--- Backups/Rob1/HOME/Module1.mod ---
MODULE Module1
!PERS tooldata DrillTool:=[TRUE,[[31.792631019,0,229.638935148],[0.945518576,0,0.325568154,0]],[1,[0,0,1],[1,0,0,0],0,0,0]];
PERS tooldata DrillTool:=[TRUE,[[67.056,0,55.372],[0.7071,0,0.7071,0]],[1,[0,0,1],[1,0,0,0],0,0,0]];
PERS wobjdata FakeWing:=[FALSE, TRUE, "",[[154, -596.9, 290],[0, 0.1326, 0, 0.9912]],[[0, 0, 0],[1, 0, 0, 0]]];
!PERS wobjdata FakeWing:=[FALSE, TRUE, "",[[154, -322.58, 290],[0,0,0,1]],[[0, 0, 0],[1, 0, 0, 0]]];
CONST jointtarget jHome:=[[-90,0,28.434410486,3.185484116,-20,-3.571881577],[9E+09,9E+09,9E+09,9E+09,9E+09,9E+09]];
	CONST robtarget Target_10:=[[25.4,-256.2,-27.8],[0.0113580960105811,-0.801870156996903,0.57220314404859,0.171635680770881],[0,0,0,1],[9E+09,9E+09,9E+09,9E+09,9E+09,9E+09]];
	CONST robtarget Target_20:=[[25.4,-251.5,-26.8],[0.00934854871281768,-0.800936484340026,0.573902636486851,0.170438013727704],[0,0,0,1],[9E+09,9E+09,9E+09,9E+09,9E+09,9E+09]];
	CONST robtarget Target_30:=[[25.4,-246.7,-25.8],[0.00738585622544953,-0.799995428854368,0.575595110655205,0.169242522817864],[0,0,0,1],[9E+09,9E+09,9E+09,9E+09,9E+09,9E+09]];
	CONST robtarget Target_40:=[[25.4,-242,-24.8],[0.00544599211880825,-0.799100144747581,0.577206071085835,0.168054905718017],[0,0,0,1],[9E+09,9E+09,9E+09,9E+09,9E+09,9E+09]];
	CONST robtarget Target_50:=[[25.4,-237.3,-23.8],[0.00347861493687028,-0.798230983744147,0.578772117197483,0.166847331964629],[0,0,0,1],[9E+09,9E+09,9E+09,9E+09,9E+09,9E+09]];
	CONST robtarget Target_60:=[[25.4,-232.5,-22.9],[0.00155774511334554,-0.797353967904281,0.580333117220716,0.165643280438256],[0,0,0,1],[9E+09,9E+09,9E+09,9E+09,9E+09,9E+09]];
	CONST robtarget Target_70:=[[25.4,-227.8,-21.9],[-0.000343161028673128,-0.796523037582201,0.581818895966585,0.164431460303543],[0,0,0,1],[9E+09,9E+09,9E+09,9E+09,9E+09,9E+09]];
	CONST robtarget Target_80:=[[25.4,-223,-21],[-0.00227982923064156,-0.795692138630642,0.58329634877276,0.163199854192462],[0,0,0,1],[9E+09,9E+09,9E+09,9E+09,9E+09,9E+09]];
	CONST robtarget Target_90:=[[25.4,-218.3,-20.1],[-0.00415671334714131,-0.794897215588351,0.584705500460769,0.161989555573681],[0,0,0,1],[9E+09,9E+09,9E+09,9E+09,9E+09,9E+09]];
	CONST robtarget Target_100:=[[25.4,-213.5,-19.2],[-0.00606983909444402,-0.794105676665045,0.586106608579309,0.160743194945786],[0,0,0,1],[9E+09,9E+09,9E+09,9E+09,9E+09,9E+09]];
	CONST robtarget Target_110:=[[25.4,-208.8,-18.4],[-0.00792422315599783,-0.793348049062693,0.587443386601589,0.159519112566011],[0,0,0,1],[9E+09,9E+09,9E+09,9E+09,9E+09,9E+09]];
	CONST robtarget Target_120:=[[25.4,-204,-17.6],[-0.00977383985694139,-0.792585828477493,0.588775847716777,0.158288274033445],[0,0,0,1],[9E+09,9E+09,9E+09,9E+09,9E+09,9E+09]];
	CONST robtarget Target_130:=[[25.4,-199.3,-16.8],[-0.0116479972262109,-0.79187063814985,0.590041679393542,0.157022397049646],[0,0,0,1],[9E+09,9E+09,9E+09,9E+09,9E+09,9E+09]];
	CONST robtarget Target_140:=[[25.4,-194.5,-16],[-0.0134775760488848,-0.791139740266602,0.591307245188397,0.155794762756806],[0,0,0,1],[9E+09,9E+09,9E+09,9E+09,9E+09,9E+09]];
	CONST robtarget Target_150:=[[25.4,-189.8,-15.2],[-0.0152917657314588,-0.790446591060719,0.592512479634857,0.154561670728084],[0,0,0,1],[9E+09,9E+09,9E+09,9E+09,9E+09,9E+09]];
	CONST robtarget Target_160:=[[25.4,-185.1,-14.4],[-0.0170965714657476,-0.789768956804693,0.593687446554438,0.153322920385096],[0,0,0,1],[9E+09,9E+09,9E+09,9E+09,9E+09,9E+09]];
	CONST robtarget Target_170:=[[25.4,-180.3,-13.7],[-0.0189383920181083,-0.7890933742209,0.594856495857871,0.152048457421108],[0,0,0,1],[9E+09,9E+09,9E+09,9E+09,9E+09,9E+09]];
	CONST robtarget Target_180:=[[25.4,-175.6,-13],[-0.0207248929133501,-0.788445598386254,0.595972909516474,0.150798900266347],[0,0,0,1],[9E+09,9E+09,9E+09,9E+09,9E+09,9E+09]];
	CONST robtarget Target_190:=[[25.4,-170.8,-12.3],[-0.0225484722456159,-0.787799513101417,0.597083852612889,0.149513766943077],[0,0,0,1],[9E+09,9E+09,9E+09,9E+09,9E+09,9E+09]];
	CONST robtarget Target_200:=[[25.4,-166.1,-11.6],[-0.0243197129064465,-0.787176744880257,0.598145161875128,0.148268975882507],[0,0,0,1],[9E+09,9E+09,9E+09,9E+09,9E+09,9E+09]];
	CONST robtarget Target_210:=[[25.4,-161.3,-11],[-0.0260874898804154,-0.78654858525833,0.5992047460239,0.147018496259117],[0,0,0,1],[9E+09,9E+09,9E+09,9E+09,9E+09,9E+09]];
	CONST robtarget Target_220:=[[25.4,-156.6,-10.3],[-0.0278809945750648,-0.78596193798026,0.600210217810398,0.145719513531353],[0,0,0,1],[9E+09,9E+09,9E+09,9E+09,9E+09,9E+09]];
	CONST robtarget Target_230:=[[25.4,-151.8,-9.7],[-0.0296325952340913,-0.785359970763115,0.601217933569803,0.144459759022046],[0,0,0,1],[9E+09,9E+09,9E+09,9E+09,9E+09,9E+09]];
	CONST robtarget Target_240:=[[25.4,-147.1,-9.1],[-0.0313751328555289,-0.784785659070614,0.602177510654819,0.143210739879962],[0,0,0,1],[9E+09,9E+09,9E+09,9E+09,9E+09,9E+09]];
	CONST robtarget Target_250:=[[25.4,-142.3,-8.5],[-0.0331524140005,-0.784214983247709,0.603132486603527,0.1419118779355],[0,0,0,1],[9E+09,9E+09,9E+09,9E+09,9E+09,9E+09]];
	CONST robtarget Target_260:=[[25.4,-137.6,-8],[-0.034877347640361,-0.783666646083767,0.604045100801052,0.140640231212982],[0,0,0,1],[9E+09,9E+09,9E+09,9E+09,9E+09,9E+09]];
	CONST robtarget Target_270:=[[25.4,-132.9,-7.4],[-0.0365986103919072,-0.783126667075213,0.604935351521993,0.139378569055698],[0,0,0,1],[9E+09,9E+09,9E+09,9E+09,9E+09,9E+09]];
	CONST robtarget Target_280:=[[25.4,-128.1,-6.9],[-0.0383577272294432,-0.782587224758595,0.605821324762428,0.138081290801936],[0,0,0,1],[9E+09,9E+09,9E+09,9E+09,9E+09,9E+09]];
	CONST robtarget Target_290:=[[25.4,-123.4,-6.4],[-0.0400656367387652,-0.782068484600279,0.606668087171559,0.136811776376679],[0,0,0,1],[9E+09,9E+09,9E+09,9E+09,9E+09,9E+09]];
	CONST robtarget Target_300:=[[25.4,-118.6,-5.9],[-0.0417706616179563,-0.781543829458959,0.607514638958406,0.135537514784141],[0,0,0,1],[9E+09,9E+09,9E+09,9E+09,9E+09,9E+09]];
	CONST robtarget Target_310:=[[25.4,-113.9,-5.4],[-0.0435063932859472,-0.781051177343454,0.608316177335671,0.134229953830614],[0,0,0,1],[9E+09,9E+09,9E+09,9E+09,9E+09,9E+09]];
	CONST robtarget Target_320:=[[25.4,-109.1,-5],[-0.0452028740439187,-0.780544008668363,0.609121417468522,0.132961834716695],[0,0,0,1],[9E+09,9E+09,9E+09,9E+09,9E+09,9E+09]];
	CONST robtarget Target_330:=[[25.4,-104.4,-4.6],[-0.046885611949136,-0.780063932790252,0.609887552842283,0.131678293731398],[0,0,0,1],[9E+09,9E+09,9E+09,9E+09,9E+09,9E+09]];
	CONST robtarget Target_340:=[[25.4,-99.6,-4.2],[-0.04861077072326,-0.779581431143657,0.610649531901286,0.130372291436634],[0,0,0,1],[9E+09,9E+09,9E+09,9E+09,9E+09,9E+09]];
	CONST robtarget Target_350:=[[25.4,-94.9,-3.8],[-0.0502864189787529,-0.779116692721743,0.611377853226394,0.129095219791102],[0,0,0,1],[9E+09,9E+09,9E+09,9E+09,9E+09,9E+09]];
	CONST robtarget Target_360:=[[25.4,-90.1,-3.4],[-0.0520001006783575,-0.778651616514941,0.612102328073387,0.127782587214575],[0,0,0,1],[9E+09,9E+09,9E+09,9E+09,9E+09,9E+09]];
	CONST robtarget Target_370:=[[25.4,-85.4,-3.1],[-0.0536646621305004,-0.778203412489929,0.612794807637811,0.126499314462914],[0,0,0,1],[9E+09,9E+09,9E+09,9E+09,9E+09,9E+09]];
	CONST robtarget Target_380:=[[25.4,-80.7,-2.7],[-0.0553238489574246,-0.77776300170738,0.613470169447094,0.125213162687542],[0,0,0,1],[9E+09,9E+09,9E+09,9E+09,9E+09,9E+09]];
	CONST robtarget Target_390:=[[25.4,-75.9,-2.4],[-0.0569860150022066,-0.77731443415222,0.614145686708351,0.123935225219912],[0,0,0,1],[9E+09,9E+09,9E+09,9E+09,9E+09,9E+09]];
	CONST robtarget Target_400:=[[25.4,-71.2,-2.1],[-0.0586751876109112,-0.776894569887548,0.614783164526675,0.122612031435063],[0,0,0,1],[9E+09,9E+09,9E+09,9E+09,9E+09,9E+09]];
	CONST robtarget Target_410:=[[25.4,-66.4,-1.9],[-0.0603271872625083,-0.776461071687208,0.615425263134368,0.121328397860276],[0,0,0,1],[9E+09,9E+09,9E+09,9E+09,9E+09,9E+09]];
	CONST robtarget Target_420:=[[25.4,-61.7,-1.6],[-0.0619717124676495,-0.776047982126195,0.616034600462907,0.120043356018546],[0,0,0,1],[9E+09,9E+09,9E+09,9E+09,9E+09,9E+09]];
	CONST robtarget Target_430:=[[25.4,-56.9,-1.4],[-0.063654337047,-0.775633930210214,0.616640125167891,0.118722734615959],[0,0,0,1],[9E+09,9E+09,9E+09,9E+09,9E+09,9E+09]];
	CONST robtarget Target_440:=[[25.4,-52.2,-1.1],[-0.0652893578640036,-0.775234130977816,0.61721871302553,0.117432543223271],[0,0,0,1],[9E+09,9E+09,9E+09,9E+09,9E+09,9E+09]];
	CONST robtarget Target_450:=[[25.4,-47.4,-0.9],[-0.0669689070708674,-0.774831453886875,0.617792784809483,0.116118295675694],[0,0,0,1],[9E+09,9E+09,9E+09,9E+09,9E+09,9E+09]];
	CONST robtarget Target_460:=[[25.4,-42.7,-0.8],[-0.0685947840793333,-0.774444127586446,0.618341874516178,0.114823233989456],[0,0,0,1],[9E+09,9E+09,9E+09,9E+09,9E+09,9E+09]];
	CONST robtarget Target_470:=[[25.4,-37.9,-0.6],[-0.0702251950846496,-0.774048910249563,0.618891208798363,0.113535801353087],[0,0,0,1],[9E+09,9E+09,9E+09,9E+09,9E+09,9E+09]];
	CONST robtarget Target_480:=[[25.4,-33.2,-0.5],[-0.0718893502838438,-0.773676551204279,0.619406337541587,0.112215437644457],[0,0,0,1],[9E+09,9E+09,9E+09,9E+09,9E+09,9E+09]];
	CONST robtarget Target_490:=[[25.4,-28.5,-0.3],[-0.0735091429764661,-0.773304826213177,0.619912706592075,0.110924694545269],[0,0,0,1],[9E+09,9E+09,9E+09,9E+09,9E+09,9E+09]];
	CONST robtarget Target_500:=[[25.4,-23.7,-0.2],[-0.0751268762924455,-0.772926904927033,0.620420125378589,0.109630379565486],[0,0,0,1],[9E+09,9E+09,9E+09,9E+09,9E+09,9E+09]];
	CONST robtarget Target_510:=[[25.4,-19,-0.2],[-0.0767785359193531,-0.772570517222499,0.620894717021794,0.108303290416625],[0,0,0,1],[9E+09,9E+09,9E+09,9E+09,9E+09,9E+09]];
	CONST robtarget Target_520:=[[25.4,-14.2,-0.1],[-0.0783956408178687,-0.772201769929318,0.621374495212959,0.107015357391473],[0,0,0,1],[9E+09,9E+09,9E+09,9E+09,9E+09,9E+09]];
	CONST robtarget Target_530:=[[25.4,-9.5,0],[-0.0799992230274888,-0.771850747246867,0.621828447919395,0.105716269550184],[0,0,0,1],[9E+09,9E+09,9E+09,9E+09,9E+09,9E+09]];
	CONST robtarget Target_540:=[[25.4,-4.7,0],[-0.0816486492100062,-0.771496504751779,0.622277235046125,0.104391972782008],[0,0,0,1],[9E+09,9E+09,9E+09,9E+09,9E+09,9E+09]];
	CONST robtarget Target_550:=[[25.4,0,0],[-0.0832525257048043,-0.77115343963232,0.622705329863117,0.103099280633186],[0,0,0,1],[9E+09,9E+09,9E+09,9E+09,9E+09,9E+09]];
	CONST robtarget Target_560:=[[30.1,0,-1.3],[-0.0836404536862687,-0.768801362660341,0.625606921371793,0.102784819941782],[0,0,0,1],[9E+09,9E+09,9E+09,9E+09,9E+09,9E+09]];
	CONST robtarget Target_570:=[[34.8,0,-2.6],[-0.0840284058612932,-0.766430934306805,0.628508693841452,0.102467905764289],[0,0,0,1],[9E+09,9E+09,9E+09,9E+09,9E+09,9E+09]];
	CONST robtarget Target_580:=[[39.5,0,-3.9],[-0.0844163267896941,-0.764042324397513,0.631410232595209,0.10214856080555],[0,0,0,1],[9E+09,9E+09,9E+09,9E+09,9E+09,9E+09]];
	CONST robtarget Target_590:=[[44.2,0,-5.1],[-0.0848041606261163,-0.761635712421235,0.634311119925615,0.101826809062296],[0,0,0,1],[9E+09,9E+09,9E+09,9E+09,9E+09,9E+09]];
	CONST robtarget Target_600:=[[49,0,-6.4],[-0.085200097924907,-0.759159511925291,0.637272618861068,0.101495753688988],[0,0,0,1],[9E+09,9E+09,9E+09,9E+09,9E+09,9E+09]];
	CONST robtarget Target_610:=[[53.7,0,-7.7],[-0.0855875837551199,-0.756717100367288,0.640170903203522,0.101169215724299],[0,0,0,1],[9E+09,9E+09,9E+09,9E+09,9E+09,9E+09]];
	CONST robtarget Target_620:=[[58.4,0,-9],[-0.0859748117230649,-0.754257287630898,0.643067258809194,0.100840351310837],[0,0,0,1],[9E+09,9E+09,9E+09,9E+09,9E+09,9E+09]];
	CONST robtarget Target_630:=[[63.1,0,-10.3],[-0.0863617247713559,-0.751780291900885,0.645961258904983,0.100509189618791],[0,0,0,1],[9E+09,9E+09,9E+09,9E+09,9E+09,9E+09]];
	CONST robtarget Target_640:=[[67.8,0,-11.6],[-0.0867482656496363,-0.7492863408784,0.648852475274426,0.100175761090643],[0,0,0,1],[9E+09,9E+09,9E+09,9E+09,9E+09,9E+09]];
	CONST robtarget Target_650:=[[72.6,0,-12.8],[-0.087142587005737,-0.746722073369839,0.651801887415907,0.0998329316070456],[0,0,0,1],[9E+09,9E+09,9E+09,9E+09,9E+09,9E+09]];
	CONST robtarget Target_660:=[[77.3,0,-14.1],[-0.0875282002573034,-0.744194584856974,0.654686165400069,0.0994950192875346],[0,0,0,1],[9E+09,9E+09,9E+09,9E+09,9E+09,9E+09]];
	CONST robtarget Target_670:=[[82,0,-15.4],[-0.0879132676563278,-0.741650886033532,0.657566360561706,0.0991549397322007],[0,0,0,1],[9E+09,9E+09,9E+09,9E+09,9E+09,9E+09]];
	CONST robtarget Target_680:=[[86.7,0,-16.7],[-0.0882977316351558,-0.739091242029488,0.660442042311056,0.098812728387569],[0,0,0,1],[9E+09,9E+09,9E+09,9E+09,9E+09,9E+09]];
	CONST robtarget Target_690:=[[91.4,0,-18],[-0.0886815346640349,-0.736515927004876,0.663312780341852,0.0984684219074372],[0,0,0,1],[9E+09,9E+09,9E+09,9E+09,9E+09,9E+09]];
	CONST robtarget Target_700:=[[96.1,0,-19.3],[-0.0890646192984286,-0.73392522401178,0.66617814498522,0.098122058134425],[0,0,0,1],[9E+09,9E+09,9E+09,9E+09,9E+09,9E+09]];
	CONST robtarget Target_710:=[[100.9,0,-20.5],[-0.0894550536127219,-0.73126382047628,0.669098483154106,0.097766242059591],[0,0,0,1],[9E+09,9E+09,9E+09,9E+09,9E+09,9E+09]];
	CONST robtarget Target_720:=[[105.6,0,-21.8],[-0.0898365113642169,-0.728642914020408,0.671951679173837,0.0974158402376966],[0,0,0,1],[9E+09,9E+09,9E+09,9E+09,9E+09,9E+09]];
	CONST robtarget Target_730:=[[110.3,0,-23.1],[-0.0902170781671603,-0.726007527181841,0.674798211150562,0.0970635024625115],[0,0,0,1],[9E+09,9E+09,9E+09,9E+09,9E+09,9E+09]];
	CONST robtarget Target_740:=[[115,0,-24.4],[-0.0905966974007335,-0.72335797710495,0.677637655576582,0.0967092711346199],[0,0,0,1],[9E+09,9E+09,9E+09,9E+09,9E+09,9E+09]];
	CONST robtarget Target_750:=[[119.7,0,-25.7],[-0.0909753127685873,-0.720694588932015,0.680469591371138,0.0963531897238861],[0,0,0,1],[9E+09,9E+09,9E+09,9E+09,9E+09,9E+09]];
	CONST robtarget Target_760:=[[119.7,-4.7,-25.7],[-0.0894964456603955,-0.720663942150709,0.680499152895289,0.097748512043658],[0,0,0,1],[9E+09,9E+09,9E+09,9E+09,9E+09,9E+09]];
	CONST robtarget Target_770:=[[119.7,-9.4,-25.7],[-0.0880162719808697,-0.720632874639458,0.680523367054942,0.0991430418519903],[0,0,0,1],[9E+09,9E+09,9E+09,9E+09,9E+09,9E+09]];
	CONST robtarget Target_780:=[[119.7,-14.2,-25.8],[-0.0865428018846856,-0.720603495890162,0.680537461381074,0.100547047742977],[0,0,0,1],[9E+09,9E+09,9E+09,9E+09,9E+09,9E+09]];
	CONST robtarget Target_790:=[[119.7,-18.9,-25.8],[-0.085059938553443,-0.720571800799192,0.680550756587509,0.101939955142535],[0,0,0,1],[9E+09,9E+09,9E+09,9E+09,9E+09,9E+09]];
	CONST robtarget Target_800:=[[119.7,-23.6,-25.9],[-0.083584041621182,-0.720538427344595,0.680557491801351,0.103342068196353],[0,0,0,1],[9E+09,9E+09,9E+09,9E+09,9E+09,9E+09]];
	CONST robtarget Target_810:=[[119.7,-28.3,-26],[-0.0821066527591594,-0.720504826362092,0.680558671847999,0.104743433847213],[0,0,0,1],[9E+09,9E+09,9E+09,9E+09,9E+09,9E+09]];
	CONST robtarget Target_820:=[[119.7,-33.1,-26.2],[-0.0806272283124645,-0.720474728202172,0.680550348761864,0.106144424614581],[0,0,0,1],[9E+09,9E+09,9E+09,9E+09,9E+09,9E+09]];
	CONST robtarget Target_830:=[[119.7,-37.8,-26.3],[-0.0791469179971094,-0.720440954411049,0.680540124134773,0.107544111979611],[0,0,0,1],[9E+09,9E+09,9E+09,9E+09,9E+09,9E+09]];
	CONST robtarget Target_840:=[[119.7,-42.5,-26.5],[-0.0776727785581285,-0.720405551888667,0.680523246637386,0.108953618871318],[0,0,0,1],[9E+09,9E+09,9E+09,9E+09,9E+09,9E+09]];
	CONST robtarget Target_850:=[[119.7,-47.2,-26.6],[-0.0761895130311405,-0.720371815338409,0.680501393526366,0.110351525493748],[0,0,0,1],[9E+09,9E+09,9E+09,9E+09,9E+09,9E+09]];
	CONST robtarget Target_860:=[[119.7,-52,-26.8],[-0.0747115228913701,-0.720340440006396,0.680468644477677,0.111759843957285],[0,0,0,1],[9E+09,9E+09,9E+09,9E+09,9E+09,9E+09]];
	CONST robtarget Target_870:=[[119.7,-56.7,-27.1],[-0.0732253755943593,-0.720307140577433,0.680434751151304,0.113155720261464],[0,0,0,1],[9E+09,9E+09,9E+09,9E+09,9E+09,9E+09]];
	CONST robtarget Target_880:=[[119.7,-61.4,-27.3],[-0.0717448887914529,-0.720272374985656,0.68039399227409,0.114561738997581],[0,0,0,1],[9E+09,9E+09,9E+09,9E+09,9E+09,9E+09]];
	CONST robtarget Target_890:=[[119.7,-66.1,-27.6],[-0.0702696329912503,-0.720236097011316,0.680346371155896,0.1159782673443],[0,0,0,1],[9E+09,9E+09,9E+09,9E+09,9E+09,9E+09]];
	CONST robtarget Target_900:=[[119.7,-70.9,-27.8],[-0.0687850809253925,-0.720206259937601,0.680288774358502,0.117382874690421],[0,0,0,1],[9E+09,9E+09,9E+09,9E+09,9E+09,9E+09]];
	CONST robtarget Target_910:=[[119.7,-75.6,-28.1],[-0.0672996627808184,-0.720172832813,0.680229181677042,0.118785969974019],[0,0,0,1],[9E+09,9E+09,9E+09,9E+09,9E+09,9E+09]];
	CONST robtarget Target_920:=[[119.7,-80.3,-28.4],[-0.0658190780270005,-0.720138044734531,0.680162517796056,0.120199812308221],[0,0,0,1],[9E+09,9E+09,9E+09,9E+09,9E+09,9E+09]];
	CONST robtarget Target_930:=[[119.7,-85,-28.8],[-0.064336655652234,-0.720103899683729,0.680089342195864,0.121612725614418],[0,0,0,1],[9E+09,9E+09,9E+09,9E+09,9E+09,9E+09]];
	CONST robtarget Target_940:=[[119.7,-89.8,-29.1],[-0.0628515923557622,-0.72007501831515,0.680004764514919,0.123025060755081],[0,0,0,1],[9E+09,9E+09,9E+09,9E+09,9E+09,9E+09]];
	CONST robtarget Target_950:=[[119.7,-94.5,-29.5],[-0.0613655083938046,-0.720042568279418,0.67991814027433,0.124435914313536],[0,0,0,1],[9E+09,9E+09,9E+09,9E+09,9E+09,9E+09]];
	CONST robtarget Target_960:=[[119.7,-99.2,-29.9],[-0.0598776216216156,-0.720011096866214,0.679824658385715,0.125845638260513],[0,0,0,1],[9E+09,9E+09,9E+09,9E+09,9E+09,9E+09]];
	CONST robtarget Target_970:=[[119.7,-103.9,-30.3],[-0.058387940861709,-0.719980723710131,0.679724196561222,0.127254164792231],[0,0,0,1],[9E+09,9E+09,9E+09,9E+09,9E+09,9E+09]];
	CONST robtarget Target_980:=[[119.7,-108.6,-30.7],[-0.0569019629309244,-0.719949270323902,0.679616191781681,0.12867418794325],[0,0,0,1],[9E+09,9E+09,9E+09,9E+09,9E+09,9E+09]];
	CONST robtarget Target_990:=[[119.7,-113.4,-31.2],[-0.0554129551896327,-0.719924020676598,0.679495748554978,0.130093568425584],[0,0,0,1],[9E+09,9E+09,9E+09,9E+09,9E+09,9E+09]];
	CONST robtarget Target_1000:=[[119.7,-118.1,-31.7],[-0.0539227905908445,-0.719895285225862,0.679373134873898,0.131511423747453],[0,0,0,1],[9E+09,9E+09,9E+09,9E+09,9E+09,9E+09]];
	CONST robtarget Target_1010:=[[119.7,-122.8,-32.2],[-0.0524305493384612,-0.7198680665055,0.679243054579513,0.132928090060728],[0,0,0,1],[9E+09,9E+09,9E+09,9E+09,9E+09,9E+09]];
	CONST robtarget Target_1020:=[[119.7,-127.5,-32.7],[-0.0509362308012004,-0.719842507181339,0.6791053603599,0.134343495477456],[0,0,0,1],[9E+09,9E+09,9E+09,9E+09,9E+09,9E+09]];
	CONST robtarget Target_1030:=[[119.7,-132.3,-33.2],[-0.0494387596832467,-0.71982411965525,0.678954212481979,0.135757957985906],[0,0,0,1],[9E+09,9E+09,9E+09,9E+09,9E+09,9E+09]];
	CONST robtarget Target_1040:=[[119.7,-137,-33.7],[-0.0479448372699026,-0.719799803937581,0.67880042479814,0.137184248820506],[0,0,0,1],[9E+09,9E+09,9E+09,9E+09,9E+09,9E+09]];
	CONST robtarget Target_1050:=[[119.7,-141.7,-34.3],[-0.0464440772866591,-0.719780190794116,0.678638852589163,0.138595571292312],[0,0,0,1],[9E+09,9E+09,9E+09,9E+09,9E+09,9E+09]];
	CONST robtarget Target_1060:=[[119.7,-146.4,-34.9],[-0.044945509749326,-0.719760119267005,0.678468776104705,0.140019254808413],[0,0,0,1],[9E+09,9E+09,9E+09,9E+09,9E+09,9E+09]];
	CONST robtarget Target_1070:=[[119.7,-151.2,-35.5],[-0.04344331380953,-0.719748215733065,0.67828412552036,0.141441965135516],[0,0,0,1],[9E+09,9E+09,9E+09,9E+09,9E+09,9E+09]];
	CONST robtarget Target_1080:=[[119.7,-155.9,-36.1],[-0.0419398630139701,-0.719733141246756,0.678096934583651,0.142862873377593],[0,0,0,1],[9E+09,9E+09,9E+09,9E+09,9E+09,9E+09]];
	CONST robtarget Target_1090:=[[119.7,-160.6,-36.8],[-0.0404378111769494,-0.719717853139121,0.677900787346707,0.144296631335408],[0,0,0,1],[9E+09,9E+09,9E+09,9E+09,9E+09,9E+09]];
	CONST robtarget Target_1100:=[[119.7,-165.3,-37.4],[-0.0389292896217268,-0.719708346409807,0.677695848544467,0.145714595642316],[0,0,0,1],[9E+09,9E+09,9E+09,9E+09,9E+09,9E+09]];
	CONST robtarget Target_1110:=[[119.7,-170.1,-38.1],[-0.0374204463715451,-0.719705234895391,0.677474850520684,0.147145886689034],[0,0,0,1],[9E+09,9E+09,9E+09,9E+09,9E+09,9E+09]];
	CONST robtarget Target_1120:=[[119.7,-174.8,-38.8],[-0.0359101121108122,-0.719699125713495,0.677251057216981,0.148575360655468],[0,0,0,1],[9E+09,9E+09,9E+09,9E+09,9E+09,9E+09]];
	CONST robtarget Target_1130:=[[119.7,-179.5,-39.6],[-0.0343969212798386,-0.719696439264827,0.677017651592734,0.150003288456814],[0,0,0,1],[9E+09,9E+09,9E+09,9E+09,9E+09,9E+09]];
	CONST robtarget Target_1140:=[[119.7,-184.2,-40.3],[-0.0328808379407684,-0.719697403969569,0.676774392615492,0.151429583357108],[0,0,0,1],[9E+09,9E+09,9E+09,9E+09,9E+09,9E+09]];
	CONST robtarget Target_1150:=[[119.7,-189,-41.1],[-0.0313227011217989,-0.719701525474739,0.676515916078243,0.152888253036598],[0,0,0,1],[9E+09,9E+09,9E+09,9E+09,9E+09,9E+09]];
	CONST robtarget Target_1160:=[[119.7,-193.7,-41.8],[-0.0298034665228329,-0.719707226208557,0.676251912667609,0.154326318364067],[0,0,0,1],[9E+09,9E+09,9E+09,9E+09,9E+09,9E+09]];
	CONST robtarget Target_1170:=[[119.7,-198.4,-42.7],[-0.0282782545443338,-0.719720645240234,0.675977312325804,0.155747251518894],[0,0,0,1],[9E+09,9E+09,9E+09,9E+09,9E+09,9E+09]];
	CONST robtarget Target_1180:=[[119.7,-203.1,-43.5],[-0.0267524651301361,-0.719735227263147,0.675691775794042,0.157181844912896],[0,0,0,1],[9E+09,9E+09,9E+09,9E+09,9E+09,9E+09]];
	CONST robtarget Target_1190:=[[119.7,-207.8,-44.3],[-0.025223237659445,-0.719754635060129,0.675395034276378,0.158614631312015],[0,0,0,1],[9E+09,9E+09,9E+09,9E+09,9E+09,9E+09]];
	CONST robtarget Target_1200:=[[119.7,-212.6,-45.2],[-0.0236886641589516,-0.719786940489491,0.675078480097401,0.160045784700893],[0,0,0,1],[9E+09,9E+09,9E+09,9E+09,9E+09,9E+09]];
	CONST robtarget Target_1210:=[[119.7,-217.3,-46.1],[-0.0221522985735409,-0.719817091465536,0.674758155864385,0.161474646915544],[0,0,0,1],[9E+09,9E+09,9E+09,9E+09,9E+09,9E+09]];
	CONST robtarget Target_1220:=[[119.7,-222,-47],[-0.0206141863419386,-0.719849213890361,0.674425687869945,0.162917636012926],[0,0,0,1],[9E+09,9E+09,9E+09,9E+09,9E+09,9E+09]];
	CONST robtarget Target_1230:=[[119.7,-226.7,-47.9],[-0.0190720397614266,-0.719887298952837,0.674080672462593,0.164358696508904],[0,0,0,1],[9E+09,9E+09,9E+09,9E+09,9E+09,9E+09]];
	CONST robtarget Target_1240:=[[119.7,-231.5,-48.8],[-0.017522051639576,-0.719944217002652,0.673713459494826,0.1657814121254],[0,0,0,1],[9E+09,9E+09,9E+09,9E+09,9E+09,9E+09]];
	CONST robtarget Target_1250:=[[119.7,-236.2,-49.8],[-0.015971633572572,-0.719995604729686,0.673341915881814,0.167218122246257],[0,0,0,1],[9E+09,9E+09,9E+09,9E+09,9E+09,9E+09]];
	CONST robtarget Target_1260:=[[119.7,-240.9,-50.8],[-0.0144181905769114,-0.72005000024701,0.672956724338874,0.168669381014636],[0,0,0,1],[9E+09,9E+09,9E+09,9E+09,9E+09,9E+09]];
	CONST robtarget Target_1270:=[[119.7,-245.6,-51.8],[-0.0128588450933917,-0.720115913737561,0.672557190492338,0.170101576717661],[0,0,0,1],[9E+09,9E+09,9E+09,9E+09,9E+09,9E+09]];
	CONST robtarget Target_1280:=[[119.7,-250.4,-52.8],[-0.0112925044941989,-0.720199272482732,0.67213276921627,0.171531419288889],[0,0,0,1],[9E+09,9E+09,9E+09,9E+09,9E+09,9E+09]];
	CONST robtarget Target_1290:=[[124.4,-250.1,-54.1],[-0.0124892710517159,-0.715646802561406,0.676985636827823,0.171417967614427],[0,0,0,1],[9E+09,9E+09,9E+09,9E+09,9E+09,9E+09]];
	CONST robtarget Target_1300:=[[129.2,-249.8,-55.3],[-0.0136732464916139,-0.710952639941439,0.681913661872113,0.171327592181889],[0,0,0,1],[9E+09,9E+09,9E+09,9E+09,9E+09,9E+09]];
	CONST robtarget Target_1310:=[[133.9,-249.5,-56.6],[-0.0148322979384848,-0.706321889232599,0.68670902664697,0.171231143342349],[0,0,0,1],[9E+09,9E+09,9E+09,9E+09,9E+09,9E+09]];
	CONST robtarget Target_1320:=[[138.6,-249.2,-57.8],[-0.0159904837570115,-0.701659547870884,0.691472181196874,0.17112687089315],[0,0,0,1],[9E+09,9E+09,9E+09,9E+09,9E+09,9E+09]];
	CONST robtarget Target_1330:=[[143.3,-248.9,-59.1],[-0.0171473278292349,-0.696967568679161,0.696201196994802,0.171014825850804],[0,0,0,1],[9E+09,9E+09,9E+09,9E+09,9E+09,9E+09]];
	CONST robtarget Target_1340:=[[148,-248.6,-60.3],[-0.0183023566454308,-0.692247946763705,0.700894199354632,0.170895070887628],[0,0,0,1],[9E+09,9E+09,9E+09,9E+09,9E+09,9E+09]];
	CONST robtarget Target_1350:=[[152.7,-248.3,-61.6],[-0.0194551004124707,-0.687502714644314,0.705549371656042,0.170767680140021],[0,0,0,1],[9E+09,9E+09,9E+09,9E+09,9E+09,9E+09]];
	CONST robtarget Target_1360:=[[157.5,-248,-62.8],[-0.020665147486378,-0.682640814131333,0.710261824935529,0.170594872726963],[0,0,0,1],[9E+09,9E+09,9E+09,9E+09,9E+09,9E+09]];
	CONST robtarget Target_1370:=[[162.2,-247.7,-64.1],[-0.0218116442228955,-0.67785006818605,0.714835383944307,0.170452078595881],[0,0,0,1],[9E+09,9E+09,9E+09,9E+09,9E+09,9E+09]];
	CONST robtarget Target_1380:=[[166.9,-247.4,-65.3],[-0.0229544688497021,-0.673040027567628,0.719366014189164,0.170301941507402],[0,0,0,1],[9E+09,9E+09,9E+09,9E+09,9E+09,9E+09]];
	CONST robtarget Target_1390:=[[171.6,-247.1,-66.6],[-0.0240931772944183,-0.668212823778592,0.723852169449314,0.170144578900482],[0,0,0,1],[9E+09,9E+09,9E+09,9E+09,9E+09,9E+09]];
	CONST robtarget Target_1400:=[[176.3,-246.8,-67.8],[-0.0252273343467782,-0.663370599750435,0.728292378420498,0.169980118023016],[0,0,0,1],[9E+09,9E+09,9E+09,9E+09,9E+09,9E+09]];
	CONST robtarget Target_1410:=[[181.1,-246.5,-69.1],[-0.0263806014436528,-0.658411567480971,0.732778649310888,0.169804955136279],[0,0,0,1],[9E+09,9E+09,9E+09,9E+09,9E+09,9E+09]];
	CONST robtarget Target_1420:=[[185.8,-246.3,-70.3],[-0.0275064663910176,-0.653536001923108,0.737130270216193,0.169626216216841],[0,0,0,1],[9E+09,9E+09,9E+09,9E+09,9E+09,9E+09]];
	CONST robtarget Target_1430:=[[190.5,-245.9,-71.6],[-0.0286561087187912,-0.648679495354103,0.741414655653978,0.169404982576479],[0,0,0,1],[9E+09,9E+09,9E+09,9E+09,9E+09,9E+09]];
	CONST robtarget Target_1440:=[[195.2,-245.7,-72.8],[-0.0297703457473825,-0.643786183416851,0.745667572952535,0.169212727661727],[0,0,0,1],[9E+09,9E+09,9E+09,9E+09,9E+09,9E+09]];
	CONST robtarget Target_1450:=[[199.9,-245.4,-74.1],[-0.0308755214603676,-0.638899471183747,0.749858816733182,0.169014564056447],[0,0,0,1],[9E+09,9E+09,9E+09,9E+09,9E+09,9E+09]];
	CONST robtarget Target_1460:=[[204.6,-245.1,-75.3],[-0.0319737541914932,-0.634010595270966,0.753996912722801,0.168810247708907],[0,0,0,1],[9E+09,9E+09,9E+09,9E+09,9E+09,9E+09]];
	CONST robtarget Target_1470:=[[209.3,-244.8,-76.6],[-0.0330646930109029,-0.629121636933686,0.758080962202085,0.168599960749507],[0,0,0,1],[9E+09,9E+09,9E+09,9E+09,9E+09,9E+09]];
	CONST robtarget Target_1480:=[[214.1,-244.5,-77.8],[-0.0341712180146319,-0.624129563242526,0.762196213319151,0.168379180862828],[0,0,0,1],[9E+09,9E+09,9E+09,9E+09,9E+09,9E+09]];
	CONST robtarget Target_1490:=[[214.1,-239.8,-76.8],[-0.0352685565372593,-0.625344750184507,0.761505650251853,0.166760957573877],[0,0,0,1],[9E+09,9E+09,9E+09,9E+09,9E+09,9E+09]];
	CONST robtarget Target_1500:=[[214.1,-235.1,-75.8],[-0.036377410933379,-0.626530843722664,0.760827103763876,0.165160237394547],[0,0,0,1],[9E+09,9E+09,9E+09,9E+09,9E+09,9E+09]];
	CONST robtarget Target_1510:=[[214.1,-230.4,-74.8],[-0.0374905350461494,-0.627696847333574,0.760160850569989,0.163543905084095],[0,0,0,1],[9E+09,9E+09,9E+09,9E+09,9E+09,9E+09]];
	CONST robtarget Target_1520:=[[214.1,-225.7,-73.9],[-0.0385817057921211,-0.628827052341548,0.759506197346856,0.161982487983516],[0,0,0,1],[9E+09,9E+09,9E+09,9E+09,9E+09,9E+09]];
	CONST robtarget Target_1530:=[[214.1,-221,-72.9],[-0.0397129990436774,-0.629943181324887,0.758861906903818,0.160384139675776],[0,0,0,1],[9E+09,9E+09,9E+09,9E+09,9E+09,9E+09]];
	CONST robtarget Target_1540:=[[214.1,-216.3,-72],[-0.0408551063250609,-0.631033669006859,0.758227646379614,0.158802409089222],[0,0,0,1],[9E+09,9E+09,9E+09,9E+09,9E+09,9E+09]];
	CONST robtarget Target_1550:=[[214.1,-211.6,-71.1],[-0.0419668302732848,-0.632098525050186,0.757604653725667,0.15724321428731],[0,0,0,1],[9E+09,9E+09,9E+09,9E+09,9E+09,9E+09]];
	CONST robtarget Target_1560:=[[214.1,-206.9,-70.2],[-0.0431220973517324,-0.633147478237495,0.756990026801105,0.155662631498866],[0,0,0,1],[9E+09,9E+09,9E+09,9E+09,9E+09,9E+09]];
	CONST robtarget Target_1570:=[[214.1,-202.2,-69.4],[-0.0442793548151249,-0.634180120150372,0.756384963217846,0.154067197550788],[0,0,0,1],[9E+09,9E+09,9E+09,9E+09,9E+09,9E+09]];
	CONST robtarget Target_1580:=[[214.1,-197.5,-68.6],[-0.0454467284791908,-0.635189863884349,0.755788257500963,0.152487840540739],[0,0,0,1],[9E+09,9E+09,9E+09,9E+09,9E+09,9E+09]];
	CONST robtarget Target_1590:=[[214.1,-192.8,-67.7],[-0.0465864465741739,-0.636172890269665,0.755201164633342,0.15094687018278],[0,0,0,1],[9E+09,9E+09,9E+09,9E+09,9E+09,9E+09]];
	CONST robtarget Target_1600:=[[214.1,-188.1,-66.9],[-0.0477695461555189,-0.63714240176872,0.754620547485047,0.149383598972081],[0,0,0,1],[9E+09,9E+09,9E+09,9E+09,9E+09,9E+09]];
	CONST robtarget Target_1610:=[[214.1,-183.4,-66.2],[-0.0489533985393246,-0.638097583939901,0.754048044913025,0.147805900099946],[0,0,0,1],[9E+09,9E+09,9E+09,9E+09,9E+09,9E+09]];
	CONST robtarget Target_1620:=[[214.1,-178.7,-65.4],[-0.0501135494154515,-0.639024535867129,0.753483945328914,0.146281300432967],[0,0,0,1],[9E+09,9E+09,9E+09,9E+09,9E+09,9E+09]];
	CONST robtarget Target_1630:=[[214.1,-174,-64.7],[-0.0513121794704837,-0.639942656609551,0.752925495500269,0.144719227178605],[0,0,0,1],[9E+09,9E+09,9E+09,9E+09,9E+09,9E+09]];
	CONST robtarget Target_1640:=[[214.1,-169.3,-64],[-0.0525156005654393,-0.640844533278809,0.752373783438205,0.143157556066027],[0,0,0,1],[9E+09,9E+09,9E+09,9E+09,9E+09,9E+09]];
	CONST robtarget Target_1650:=[[214.1,-164.6,-63.3],[-0.0536899475070816,-0.641723004287069,0.751830248201575,0.141634223246443],[0,0,0,1],[9E+09,9E+09,9E+09,9E+09,9E+09,9E+09]];
	CONST robtarget Target_1660:=[[214.1,-159.9,-62.6],[-0.0549022874737579,-0.642593676162974,0.751291241769304,0.140073467245733],[0,0,0,1],[9E+09,9E+09,9E+09,9E+09,9E+09,9E+09]];
	CONST robtarget Target_1670:=[[214.1,-155.2,-61.9],[-0.0561242209793799,-0.643446414332673,0.750757651605653,0.138527009126195],[0,0,0,1],[9E+09,9E+09,9E+09,9E+09,9E+09,9E+09]];
	CONST robtarget Target_1680:=[[214.1,-150.4,-61.3],[-0.0573428290888,-0.644298492896021,0.750220650493769,0.136967980114748],[0,0,0,1],[9E+09,9E+09,9E+09,9E+09,9E+09,9E+09]];
	CONST robtarget Target_1690:=[[214.1,-145.7,-60.7],[-0.0585391714057714,-0.64511482893062,0.749700327915236,0.135460109363351],[0,0,0,1],[9E+09,9E+09,9E+09,9E+09,9E+09,9E+09]];
	CONST robtarget Target_1700:=[[214.1,-141,-60.1],[-0.0597731615365629,-0.645924637221304,0.749183165378491,0.133914588092245],[0,0,0,1],[9E+09,9E+09,9E+09,9E+09,9E+09,9E+09]];
	CONST robtarget Target_1710:=[[214.1,-136.3,-59.5],[-0.0610108478057296,-0.646720866963663,0.748670915845893,0.132369393933289],[0,0,0,1],[9E+09,9E+09,9E+09,9E+09,9E+09,9E+09]];
	CONST robtarget Target_1720:=[[214.1,-131.6,-59],[-0.0622181375236594,-0.647496731507395,0.748165675952307,0.13086255146968],[0,0,0,1],[9E+09,9E+09,9E+09,9E+09,9E+09,9E+09]];
	CONST robtarget Target_1730:=[[214.1,-126.9,-58.4],[-0.0634688183068436,-0.648264268897657,0.747662116568994,0.129330994819074],[0,0,0,1],[9E+09,9E+09,9E+09,9E+09,9E+09,9E+09]];
	CONST robtarget Target_1740:=[[214.1,-122.3,-57.9],[-0.064724629163582,-0.649009411435852,0.747171328797483,0.127798715448665],[0,0,0,1],[9E+09,9E+09,9E+09,9E+09,9E+09,9E+09]];
	CONST robtarget Target_1750:=[[214.1,-117.6,-57.4],[-0.0659415982702471,-0.649747743117887,0.746679097173527,0.126292920525678],[0,0,0,1],[9E+09,9E+09,9E+09,9E+09,9E+09,9E+09]];
	CONST robtarget Target_1760:=[[214.1,-112.9,-56.9],[-0.0672019671558274,-0.650478513802981,0.746187667457493,0.12476202797886],[0,0,0,1],[9E+09,9E+09,9E+09,9E+09,9E+09,9E+09]];
	CONST robtarget Target_1770:=[[214.1,-108.1,-56.5],[-0.0684638092553564,-0.65120670448846,0.745691861757032,0.123232228580258],[0,0,0,1],[9E+09,9E+09,9E+09,9E+09,9E+09,9E+09]];
	CONST robtarget Target_1780:=[[214.1,-103.4,-56.1],[-0.0697368456344226,-0.651911675562493,0.745207121516542,0.121713950175375],[0,0,0,1],[9E+09,9E+09,9E+09,9E+09,9E+09,9E+09]];
	CONST robtarget Target_1790:=[[214.1,-98.7,-55.6],[-0.0709718230450671,-0.652600969502751,0.744729273860509,0.120221809971935],[0,0,0,1],[9E+09,9E+09,9E+09,9E+09,9E+09,9E+09]];
	CONST robtarget Target_1800:=[[214.1,-94,-55.2],[-0.0722505034042859,-0.653283696519975,0.744251094825556,0.118703767716048],[0,0,0,1],[9E+09,9E+09,9E+09,9E+09,9E+09,9E+09]];
	CONST robtarget Target_1810:=[[214.1,-89.3,-54.9],[-0.073531882239943,-0.653955613371436,0.743775907688082,0.117185823276578],[0,0,0,1],[9E+09,9E+09,9E+09,9E+09,9E+09,9E+09]];
	CONST robtarget Target_1820:=[[214.1,-84.6,-54.5],[-0.0747816180925732,-0.654610534044765,0.743306705241576,0.115706094290646],[0,0,0,1],[9E+09,9E+09,9E+09,9E+09,9E+09,9E+09]];
	CONST robtarget Target_1830:=[[214.1,-79.9,-54.2],[-0.0760679807605466,-0.65526150182537,0.742837140883982,0.114188478630225],[0,0,0,1],[9E+09,9E+09,9E+09,9E+09,9E+09,9E+09]];
	CONST robtarget Target_1840:=[[214.1,-75.2,-53.8],[-0.0773566576912869,-0.655902245050804,0.742370135670044,0.112671088187645],[0,0,0,1],[9E+09,9E+09,9E+09,9E+09,9E+09,9E+09]];
	CONST robtarget Target_1850:=[[214.1,-70.5,-53.5],[-0.0786209131429899,-0.656524923359305,0.741908117772246,0.111203065642386],[0,0,0,1],[9E+09,9E+09,9E+09,9E+09,9E+09,9E+09]];
	CONST robtarget Target_1860:=[[214.1,-65.8,-53.3],[-0.0799139638073097,-0.657145878750976,0.741445892179642,0.10968610394734],[0,0,0,1],[9E+09,9E+09,9E+09,9E+09,9E+09,9E+09]];
	CONST robtarget Target_1870:=[[214.1,-61.1,-53],[-0.0812168877925794,-0.657755387238009,0.74098496061655,0.108180200761296],[0,0,0,1],[9E+09,9E+09,9E+09,9E+09,9E+09,9E+09]];
	CONST robtarget Target_1880:=[[214.1,-56.4,-52.8],[-0.0825219107000369,-0.658355458149378,0.740526028980437,0.10667438953096],[0,0,0,1],[9E+09,9E+09,9E+09,9E+09,9E+09,9E+09]];
	CONST robtarget Target_1890:=[[214.1,-51.7,-52.5],[-0.0837945760408972,-0.658940359613963,0.740072696951967,0.105206818810331],[0,0,0,1],[9E+09,9E+09,9E+09,9E+09,9E+09,9E+09]];
	CONST robtarget Target_1900:=[[214.1,-47,-52.3],[-0.0851034431169612,-0.659522090614642,0.739617502834651,0.103701328157192],[0,0,0,1],[9E+09,9E+09,9E+09,9E+09,9E+09,9E+09]];
	CONST robtarget Target_1910:=[[214.1,-42.3,-52.1],[-0.0864225230900232,-0.660093279955253,0.739162979927188,0.102206156203186],[0,0,0,1],[9E+09,9E+09,9E+09,9E+09,9E+09,9E+09]];
	CONST robtarget Target_1920:=[[214.1,-37.6,-52],[-0.0877005611737851,-0.660651556753741,0.73871493975808,0.10073911805688],[0,0,0,1],[9E+09,9E+09,9E+09,9E+09,9E+09,9E+09]];
	CONST robtarget Target_1930:=[[214.1,-32.9,-51.8],[-0.0890232355278324,-0.661205404795119,0.738263427899601,0.0992440790768353],[0,0,0,1],[9E+09,9E+09,9E+09,9E+09,9E+09,9E+09]];
	CONST robtarget Target_1940:=[[214.1,-28.2,-51.7],[-0.0903476248802413,-0.66175076707453,0.737813216726165,0.0977490980979308],[0,0,0,1],[9E+09,9E+09,9E+09,9E+09,9E+09,9E+09]];
	CONST robtarget Target_1950:=[[214.1,-23.5,-51.6],[-0.0916392101554855,-0.662282314080756,0.737368414746666,0.0962923286243821],[0,0,0,1],[9E+09,9E+09,9E+09,9E+09,9E+09,9E+09]];
	CONST robtarget Target_1960:=[[214.1,-18.8,-51.5],[-0.0929667151175744,-0.662811152057207,0.736920607127253,0.0947976021851103],[0,0,0,1],[9E+09,9E+09,9E+09,9E+09,9E+09,9E+09]];
	CONST robtarget Target_1970:=[[214.1,-14.1,-51.4],[-0.0943048826559268,-0.663330579630775,0.736472643001956,0.093312257199492],[0,0,0,1],[9E+09,9E+09,9E+09,9E+09,9E+09,9E+09]];
	CONST robtarget Target_1980:=[[214.1,-9.4,-51.4],[-0.0956352507820257,-0.663843336202951,0.73602677354098,0.0918178218955898],[0,0,0,1],[9E+09,9E+09,9E+09,9E+09,9E+09,9E+09]];
	CONST robtarget Target_1990:=[[214.1,-4.7,-51.4],[-0.0969419126319893,-0.664341826293298,0.735585037755558,0.0903706569783089],[0,0,0,1],[9E+09,9E+09,9E+09,9E+09,9E+09,9E+09]];
	CONST robtarget Target_2000:=[[214.1,0,-51.4],[-0.0982844100354686,-0.664837850533483,0.735139570282207,0.0888854287681022],[0,0,0,1],[9E+09,9E+09,9E+09,9E+09,9E+09,9E+09]];
	CONST robtarget Target_2010:=[[218.8,0,-52.6],[-0.0986298157811465,-0.661969917710996,0.737723107501987,0.0885020007812625],[0,0,0,1],[9E+09,9E+09,9E+09,9E+09,9E+09,9E+09]];
	CONST robtarget Target_2020:=[[223.5,0,-53.9],[-0.0989731463768498,-0.659096812484189,0.740291123187272,0.0881178812703537],[0,0,0,1],[9E+09,9E+09,9E+09,9E+09,9E+09,9E+09]];
	CONST robtarget Target_2030:=[[228.2,0,-55.2],[-0.0993143645339152,-0.656218964864421,0.742843338429415,0.0877331277257005],[0,0,0,1],[9E+09,9E+09,9E+09,9E+09,9E+09,9E+09]];
	CONST robtarget Target_2040:=[[232.9,0,-56.5],[-0.0996534341613626,-0.653336805334557,0.745379483278099,0.0873477977006659],[0,0,0,1],[9E+09,9E+09,9E+09,9E+09,9E+09,9E+09]];
	CONST robtarget Target_2050:=[[237.6,0,-57.8],[-0.0999903203834938,-0.650450764496132,0.747899296872973,0.0869619487644783],[0,0,0,1],[9E+09,9E+09,9E+09,9E+09,9E+09,9E+09]];
	CONST robtarget Target_2060:=[[242.4,0,-59.1],[-0.100332085849476,-0.647499759825167,0.750455605830912,0.0865674144953103],[0,0,0,1],[9E+09,9E+09,9E+09,9E+09,9E+09,9E+09]];
	CONST robtarget Target_2070:=[[247.1,0,-60.3],[-0.100664457368582,-0.644607187285649,0.752941650724925,0.0861806923040096],[0,0,0,1],[9E+09,9E+09,9E+09,9E+09,9E+09,9E+09]];
	CONST robtarget Target_2080:=[[251.8,0,-61.6],[-0.100994547646667,-0.641712031583591,0.755410632581744,0.0857936247570562],[0,0,0,1],[9E+09,9E+09,9E+09,9E+09,9E+09,9E+09]];
	CONST robtarget Target_2090:=[[256.5,0,-62.9],[-0.101322326835638,-0.638814720301352,0.757862328146079,0.0854062690200298],[0,0,0,1],[9E+09,9E+09,9E+09,9E+09,9E+09,9E+09]];
	CONST robtarget Target_2100:=[[261.2,0,-64.2],[-0.10164776636341,-0.635915679422987,0.760296523706831,0.0850186820448252],[0,0,0,1],[9E+09,9E+09,9E+09,9E+09,9E+09,9E+09]];
	CONST robtarget Target_2110:=[[265.9,0,-65.5],[-0.101970838940531,-0.633015333007546,0.762713015146612,0.0846309205259742],[0,0,0,1],[9E+09,9E+09,9E+09,9E+09,9E+09,9E+09]];
	CONST robtarget Target_2120:=[[270.7,0,-66.8],[-0.102298315353963,-0.63005236804054,0.76516244603561,0.0842347872262443],[0,0,0,1],[9E+09,9E+09,9E+09,9E+09,9E+09,9E+09]];
	CONST robtarget Target_2130:=[[275.4,0,-68.1],[-0.102616525615677,-0.62715066808584,0.767542568732298,0.0838468447460998],[0,0,0,1],[9E+09,9E+09,9E+09,9E+09,9E+09,9E+09]];
	CONST robtarget Target_2140:=[[280.1,0,-69.3],[-0.102932294309493,-0.624248928879364,0.769904429192128,0.0834588970181931],[0,0,0,1],[9E+09,9E+09,9E+09,9E+09,9E+09,9E+09]];
	CONST robtarget Target_2150:=[[284.8,0,-70.6],[-0.10324559933483,-0.621347563578349,0.772247862109012,0.083070999279539],[0,0,0,1],[9E+09,9E+09,9E+09,9E+09,9E+09,9E+09]];
	CONST robtarget Target_2160:=[[289.5,0,-71.9],[-0.103556419880537,-0.618446981881466,0.774572711821425,0.0826832063047595],[0,0,0,1],[9E+09,9E+09,9E+09,9E+09,9E+09,9E+09]];
	CONST robtarget Target_2170:=[[294.2,0,-73.2],[-0.103864736421198,-0.615547589747956,0.776878832284786,0.0822955723685342],[0,0,0,1],[9E+09,9E+09,9E+09,9E+09,9E+09,9E+09]];
	CONST robtarget Target_2180:=[[299,0,-74.5],[-0.104177009443503,-0.612588154003657,0.779214546111071,0.0818999109078748],[0,0,0,1],[9E+09,9E+09,9E+09,9E+09,9E+09,9E+09]];
	CONST robtarget Target_2190:=[[303.7,0,-75.8],[-0.104480210311745,-0.609692389178512,0.781482402792595,0.0815127619242722],[0,0,0,1],[9E+09,9E+09,9E+09,9E+09,9E+09,9E+09]];
	CONST robtarget Target_2200:=[[308.4,0,-77],[-0.104780855932186,-0.606799015001593,0.783731146943764,0.0811259325581408],[0,0,0,1],[9E+09,9E+09,9E+09,9E+09,9E+09,9E+09]];
	CONST robtarget Target_2210:=[[308.4,-4.8,-77.1],[-0.10357270922086,-0.605804769828204,0.784497151639023,0.0826891397240769],[0,0,0,1],[9E+09,9E+09,9E+09,9E+09,9E+09,9E+09]];
	CONST robtarget Target_2220:=[[308.4,-9.6,-77.1],[-0.102337196398047,-0.604789512357301,0.785271515729608,0.0842934787497215],[0,0,0,1],[9E+09,9E+09,9E+09,9E+09,9E+09,9E+09]];
	CONST robtarget Target_2230:=[[308.4,-14.3,-77.1],[-0.101145369475392,-0.603779543049934,0.78603214142339,0.0858682145934034],[0,0,0,1],[9E+09,9E+09,9E+09,9E+09,9E+09,9E+09]];
	CONST robtarget Target_2240:=[[308.4,-19.1,-77.2],[-0.0999593935484523,-0.602737043222909,0.786810116681356,0.0874415041968199],[0,0,0,1],[9E+09,9E+09,9E+09,9E+09,9E+09,9E+09]];
	CONST robtarget Target_2250:=[[308.4,-23.9,-77.3],[-0.0987679840357655,-0.601679444358616,0.787594150307987,0.0890066624835305],[0,0,0,1],[9E+09,9E+09,9E+09,9E+09,9E+09,9E+09]];
	CONST robtarget Target_2260:=[[308.4,-28.6,-77.4],[-0.0975887713076906,-0.600621452045473,0.788368560100788,0.0905832020964815],[0,0,0,1],[9E+09,9E+09,9E+09,9E+09,9E+09,9E+09]];
	CONST robtarget Target_2270:=[[308.4,-33.4,-77.5],[-0.0963848720850105,-0.599523263975145,0.789164862941784,0.0921988692111749],[0,0,0,1],[9E+09,9E+09,9E+09,9E+09,9E+09,9E+09]];
	CONST robtarget Target_2280:=[[308.4,-38.2,-77.7],[-0.095226295927332,-0.59841215591312,0.789961700481073,0.0937835592863895],[0,0,0,1],[9E+09,9E+09,9E+09,9E+09,9E+09,9E+09]];
	CONST robtarget Target_2290:=[[308.4,-43,-77.9],[-0.09406320670459,-0.597284763534262,0.790765182273869,0.0953595873399466],[0,0,0,1],[9E+09,9E+09,9E+09,9E+09,9E+09,9E+09]];
	CONST robtarget Target_2300:=[[308.4,-47.7,-78.1],[-0.0929120064575001,-0.59615659109678,0.791559096194288,0.0969477961584996],[0,0,0,1],[9E+09,9E+09,9E+09,9E+09,9E+09,9E+09]];
	CONST robtarget Target_2310:=[[308.4,-52.5,-78.3],[-0.0917370265888429,-0.594985280908352,0.792376012395457,0.0985752932297051],[0,0,0,1],[9E+09,9E+09,9E+09,9E+09,9E+09,9E+09]];
	CONST robtarget Target_2320:=[[308.4,-57.3,-78.5],[-0.090598384829287,-0.593801259372321,0.793195720509647,0.100162597806529],[0,0,0,1],[9E+09,9E+09,9E+09,9E+09,9E+09,9E+09]];
	CONST robtarget Target_2330:=[[308.4,-62.1,-78.8],[-0.0894651742912847,-0.592598007640244,0.794021679272131,0.101750463270237],[0,0,0,1],[9E+09,9E+09,9E+09,9E+09,9E+09,9E+09]];
	CONST robtarget Target_2340:=[[308.4,-66.8,-79],[-0.0883349732594255,-0.591395261296902,0.794839102742081,0.103341076861959],[0,0,0,1],[9E+09,9E+09,9E+09,9E+09,9E+09,9E+09]];
	CONST robtarget Target_2350:=[[308.4,-71.6,-79.3],[-0.0872216407657374,-0.590150908215717,0.795676956264462,0.104940326776786],[0,0,0,1],[9E+09,9E+09,9E+09,9E+09,9E+09,9E+09]];
	CONST robtarget Target_2360:=[[308.4,-76.4,-79.7],[-0.0860832915980205,-0.588879448289243,0.79652439224517,0.106581212456363],[0,0,0,1],[9E+09,9E+09,9E+09,9E+09,9E+09,9E+09]];
	CONST robtarget Target_2370:=[[308.4,-81.1,-80],[-0.0849789502106103,-0.587614708040441,0.797360470344529,0.108184163571205],[0,0,0,1],[9E+09,9E+09,9E+09,9E+09,9E+09,9E+09]];
	CONST robtarget Target_2380:=[[308.4,-85.9,-80.4],[-0.0838836319156044,-0.586307668086254,0.798219267880476,0.109785495509485],[0,0,0,1],[9E+09,9E+09,9E+09,9E+09,9E+09,9E+09]];
	CONST robtarget Target_2390:=[[308.4,-90.7,-80.7],[-0.082794767336965,-0.584978717113686,0.799085584538455,0.11138741225327],[0,0,0,1],[9E+09,9E+09,9E+09,9E+09,9E+09,9E+09]];
	CONST robtarget Target_2400:=[[308.4,-95.5,-81.1],[-0.0816819800067539,-0.58362055263885,0.799961961293307,0.11303081510573],[0,0,0,1],[9E+09,9E+09,9E+09,9E+09,9E+09,9E+09]];
	CONST robtarget Target_2410:=[[308.4,-100.2,-81.5],[-0.0806113427211271,-0.582266960029181,0.800826422485906,0.114647458460705],[0,0,0,1],[9E+09,9E+09,9E+09,9E+09,9E+09,9E+09]];
	CONST robtarget Target_2420:=[[308.4,-105,-82],[-0.0795508130991443,-0.58086741275938,0.80171549259436,0.116262572927284],[0,0,0,1],[9E+09,9E+09,9E+09,9E+09,9E+09,9E+09]];
	CONST robtarget Target_2430:=[[308.4,-109.8,-82.4],[-0.0784974683762196,-0.579443805115183,0.802613049576641,0.117878398451314],[0,0,0,1],[9E+09,9E+09,9E+09,9E+09,9E+09,9E+09]];
	CONST robtarget Target_2440:=[[308.4,-114.5,-82.9],[-0.0774479655214412,-0.578019762866521,0.803501948900264,0.119497215389307],[0,0,0,1],[9E+09,9E+09,9E+09,9E+09,9E+09,9E+09]];
	CONST robtarget Target_2450:=[[308.4,-119.3,-83.4],[-0.076379344448792,-0.576539662649598,0.804418795175791,0.121155334597319],[0,0,0,1],[9E+09,9E+09,9E+09,9E+09,9E+09,9E+09]];
	CONST robtarget Target_2460:=[[308.4,-124.1,-84],[-0.075356372668175,-0.575038428608826,0.805342168587324,0.122785236150173],[0,0,0,1],[9E+09,9E+09,9E+09,9E+09,9E+09,9E+09]];
	CONST robtarget Target_2470:=[[308.4,-128.9,-84.5],[-0.0743414376682748,-0.573510671613807,0.806275092793661,0.124415975385267],[0,0,0,1],[9E+09,9E+09,9E+09,9E+09,9E+09,9E+09]];
	CONST robtarget Target_2480:=[[308.4,-133.6,-85.1],[-0.0733236228418459,-0.571984445986194,0.807200120771844,0.126037315542401],[0,0,0,1],[9E+09,9E+09,9E+09,9E+09,9E+09,9E+09]];
	CONST robtarget Target_2490:=[[308.4,-138.4,-85.7],[-0.0722955709467476,-0.570394869197485,0.808154117550502,0.127710476864027],[0,0,0,1],[9E+09,9E+09,9E+09,9E+09,9E+09,9E+09]];
	CONST robtarget Target_2500:=[[308.4,-143.2,-86.3],[-0.0713134460058373,-0.568781437267891,0.809116215699097,0.129356169280855],[0,0,0,1],[9E+09,9E+09,9E+09,9E+09,9E+09,9E+09]];
	CONST robtarget Target_2510:=[[308.4,-148,-86.9],[-0.0703335262208272,-0.567141407219054,0.81008981098623,0.130989760833546],[0,0,0,1],[9E+09,9E+09,9E+09,9E+09,9E+09,9E+09]];
	CONST robtarget Target_2520:=[[308.4,-152.7,-87.5],[-0.0693652484196903,-0.56549690491479,0.811053916248892,0.132639578485468],[0,0,0,1],[9E+09,9E+09,9E+09,9E+09,9E+09,9E+09]];
	CONST robtarget Target_2530:=[[308.4,-157.5,-88.2],[-0.0684111361139451,-0.563793801471881,0.812048792395899,0.134287842509463],[0,0,0,1],[9E+09,9E+09,9E+09,9E+09,9E+09,9E+09]];
	CONST robtarget Target_2540:=[[308.4,-162.3,-88.9],[-0.0674308680514497,-0.562054271273655,0.813057035081266,0.135964450801413],[0,0,0,1],[9E+09,9E+09,9E+09,9E+09,9E+09,9E+09]];
	CONST robtarget Target_2550:=[[308.4,-167,-89.6],[-0.0664986814080785,-0.560314130241802,0.814053991763236,0.137630299413684],[0,0,0,1],[9E+09,9E+09,9E+09,9E+09,9E+09,9E+09]];
	CONST robtarget Target_2560:=[[308.4,-171.8,-90.3],[-0.0655756202077783,-0.558514111134058,0.815084460660975,0.139280823114688],[0,0,0,1],[9E+09,9E+09,9E+09,9E+09,9E+09,9E+09]];
	CONST robtarget Target_2570:=[[308.4,-176.6,-91.1],[-0.0646636661456529,-0.55667986221951,0.816127636032455,0.14093197999016],[0,0,0,1],[9E+09,9E+09,9E+09,9E+09,9E+09,9E+09]];
	CONST robtarget Target_2580:=[[308.4,-181.4,-91.9],[-0.0637401055078415,-0.554799250276008,0.817183626452998,0.142639095272496],[0,0,0,1],[9E+09,9E+09,9E+09,9E+09,9E+09,9E+09]];
	CONST robtarget Target_2590:=[[308.4,-186.1,-92.7],[-0.0628518580764369,-0.552923084824419,0.818230272116942,0.144308447417405],[0,0,0,1],[9E+09,9E+09,9E+09,9E+09,9E+09,9E+09]];
	CONST robtarget Target_2600:=[[308.4,-190.9,-93.5],[-0.0619813474792873,-0.550977563261577,0.819312528367716,0.145976087790734],[0,0,0,1],[9E+09,9E+09,9E+09,9E+09,9E+09,9E+09]];
	CONST robtarget Target_2610:=[[308.4,-195.7,-94.3],[-0.0611233995693708,-0.548993739703088,0.820408994029005,0.147644459117901],[0,0,0,1],[9E+09,9E+09,9E+09,9E+09,9E+09,9E+09]];
	CONST robtarget Target_2620:=[[308.4,-200.4,-95.2],[-0.0602779418746451,-0.54700204307425,0.821495947228052,0.149330985678924],[0,0,0,1],[9E+09,9E+09,9E+09,9E+09,9E+09,9E+09]];
	CONST robtarget Target_2630:=[[308.4,-205.2,-96.1],[-0.0594173744366705,-0.544930762338883,0.822621633890505,0.151042005174497],[0,0,0,1],[9E+09,9E+09,9E+09,9E+09,9E+09,9E+09]];
	CONST robtarget Target_2640:=[[308.4,-210,-97],[-0.0586053434674626,-0.542822347677266,0.823761847214398,0.15272763879902],[0,0,0,1],[9E+09,9E+09,9E+09,9E+09,9E+09,9E+09]];
	CONST robtarget Target_2650:=[[308.4,-214.8,-97.9],[-0.0578075887797071,-0.540670882363083,0.824917917993721,0.154414080371918],[0,0,0,1],[9E+09,9E+09,9E+09,9E+09,9E+09,9E+09]];
	CONST robtarget Target_2660:=[[308.4,-219.5,-98.8],[-0.0570173734934169,-0.538513452607028,0.826065282156528,0.156103908012666],[0,0,0,1],[9E+09,9E+09,9E+09,9E+09,9E+09,9E+09]];
	CONST robtarget Target_2670:=[[308.4,-224.3,-99.8],[-0.05622658655833,-0.536260517000348,0.827252679079179,0.157848768848032],[0,0,0,1],[9E+09,9E+09,9E+09,9E+09,9E+09,9E+09]];
	CONST robtarget Target_2680:=[[308.4,-229.1,-100.8],[-0.0554746070084852,-0.533972825784062,0.828458451488987,0.159537404573058],[0,0,0,1],[9E+09,9E+09,9E+09,9E+09,9E+09,9E+09]];
	CONST robtarget Target_2690:=[[308.4,-233.9,-101.8],[-0.0547443984118989,-0.531632628929442,0.829681024354622,0.161242663479473],[0,0,0,1],[9E+09,9E+09,9E+09,9E+09,9E+09,9E+09]];
	CONST robtarget Target_2700:=[[308.4,-238.6,-102.8],[-0.0540228184989099,-0.529284468395526,0.830894888909729,0.162951435036297],[0,0,0,1],[9E+09,9E+09,9E+09,9E+09,9E+09,9E+09]];
	CONST robtarget Target_2710:=[[313.1,-238.3,-104.1],[-0.0548938197151421,-0.524831687057051,0.83371461853676,0.162660086241327],[0,0,0,1],[9E+09,9E+09,9E+09,9E+09,9E+09,9E+09]];
	CONST robtarget Target_2720:=[[317.8,-238,-105.3],[-0.0557536487314289,-0.520413347981774,0.836479714125481,0.162367378965379],[0,0,0,1],[9E+09,9E+09,9E+09,9E+09,9E+09,9E+09]];
	CONST robtarget Target_2730:=[[322.6,-237.7,-106.6],[-0.0566207915154303,-0.515934486926424,0.839249647066362,0.162067026464734],[0,0,0,1],[9E+09,9E+09,9E+09,9E+09,9E+09,9E+09]];
	CONST robtarget Target_2740:=[[327.3,-237.4,-107.8],[-0.0574580480235626,-0.511588011684228,0.841906212830161,0.161772086023135],[0,0,0,1],[9E+09,9E+09,9E+09,9E+09,9E+09,9E+09]];
	CONST robtarget Target_2750:=[[332,-237.2,-109.1],[-0.0582930745636434,-0.507231486237791,0.844538089294999,0.161473070686329],[0,0,0,1],[9E+09,9E+09,9E+09,9E+09,9E+09,9E+09]];
	CONST robtarget Target_2760:=[[336.7,-236.9,-110.3],[-0.0591348869443182,-0.502966637218313,0.847091105604348,0.161134371868289],[0,0,0,1],[9E+09,9E+09,9E+09,9E+09,9E+09,9E+09]];
	CONST robtarget Target_2770:=[[341.4,-236.6,-111.6],[-0.0599386765830767,-0.49873093242915,0.849591805743821,0.160837109215425],[0,0,0,1],[9E+09,9E+09,9E+09,9E+09,9E+09,9E+09]];
	CONST robtarget Target_2780:=[[346.1,-236.3,-112.8],[-0.060731418488601,-0.4945335001632,0.852041898362416,0.160539451412005],[0,0,0,1],[9E+09,9E+09,9E+09,9E+09,9E+09,9E+09]];
	CONST robtarget Target_2790:=[[350.9,-236,-114.1],[-0.0615302743962089,-0.490283545755737,0.854494484540349,0.160234971164326],[0,0,0,1],[9E+09,9E+09,9E+09,9E+09,9E+09,9E+09]];
	CONST robtarget Target_2800:=[[355.6,-235.7,-115.3],[-0.0623008583262713,-0.4861647259849,0.856844582498321,0.159936936644151],[0,0,0,1],[9E+09,9E+09,9E+09,9E+09,9E+09,9E+09]];
	CONST robtarget Target_2810:=[[360.3,-235.4,-116.6],[-0.0630800791216334,-0.482098034826904,0.859148732661681,0.159580210552165],[0,0,0,1],[9E+09,9E+09,9E+09,9E+09,9E+09,9E+09]];
	CONST robtarget Target_2820:=[[365,-235.1,-117.8],[-0.0638287234838022,-0.478058420378277,0.861403045457561,0.159282246469257],[0,0,0,1],[9E+09,9E+09,9E+09,9E+09,9E+09,9E+09]];
	CONST robtarget Target_2830:=[[369.7,-234.8,-119.1],[-0.0645666547616862,-0.4740588151663,0.863610618149904,0.158984549798872],[0,0,0,1],[9E+09,9E+09,9E+09,9E+09,9E+09,9E+09]];
	CONST robtarget Target_2840:=[[374.4,-234.5,-120.3],[-0.0652939577196355,-0.470099429006276,0.865772248842678,0.158687236623401],[0,0,0,1],[9E+09,9E+09,9E+09,9E+09,9E+09,9E+09]];
	CONST robtarget Target_2850:=[[379.1,-234.2,-121.6],[-0.0660107222946255,-0.466180430729295,0.867888740578644,0.158390418030911],[0,0,0,1],[9E+09,9E+09,9E+09,9E+09,9E+09,9E+09]];
	CONST robtarget Target_2860:=[[383.9,-233.9,-122.8],[-0.0667325868025735,-0.462216412519589,0.870006349411116,0.158087639746129],[0,0,0,1],[9E+09,9E+09,9E+09,9E+09,9E+09,9E+09]];
	CONST robtarget Target_2870:=[[388.6,-233.6,-124.1],[-0.0674528456392701,-0.45838793454485,0.872035529794928,0.157748692083801],[0,0,0,1],[9E+09,9E+09,9E+09,9E+09,9E+09,9E+09]];
	CONST robtarget Target_2880:=[[393.3,-233.3,-125.3],[-0.0681381776210262,-0.454591556613989,0.874020583519796,0.157453882103525],[0,0,0,1],[9E+09,9E+09,9E+09,9E+09,9E+09,9E+09]];
	CONST robtarget Target_2890:=[[398,-233,-126.6],[-0.0688133787721291,-0.45083586868829,0.875963745405648,0.157159966724827],[0,0,0,1],[9E+09,9E+09,9E+09,9E+09,9E+09,9E+09]];
	CONST robtarget Target_2900:=[[402.8,-232.7,-127.8],[-0.0694932440832772,-0.447038675961153,0.877907675075184,0.156860528067985],[0,0,0,1],[9E+09,9E+09,9E+09,9E+09,9E+09,9E+09]];
	CONST robtarget Target_2910:=[[402.8,-228,-126.8],[-0.069975286563823,-0.450045871985816,0.87664655423895,0.155090268294995],[0,0,0,1],[9E+09,9E+09,9E+09,9E+09,9E+09,9E+09]];
	CONST robtarget Target_2920:=[[402.8,-223.2,-125.8],[-0.0704667749223318,-0.453055520723769,0.875366669396911,0.153324241014652],[0,0,0,1],[9E+09,9E+09,9E+09,9E+09,9E+09,9E+09]];
	CONST robtarget Target_2930:=[[402.8,-218.5,-124.8],[-0.070993348790441,-0.455955857807755,0.874123011714268,0.15156899600476],[0,0,0,1],[9E+09,9E+09,9E+09,9E+09,9E+09,9E+09]];
	CONST robtarget Target_2940:=[[402.8,-213.7,-123.9],[-0.0715219932106716,-0.458862710635186,0.872862376511288,0.149802833573901],[0,0,0,1],[9E+09,9E+09,9E+09,9E+09,9E+09,9E+09]];
	CONST robtarget Target_2950:=[[402.8,-209,-122.9],[-0.0720842834673668,-0.461664617479993,0.871637303280222,0.148047453792459],[0,0,0,1],[9E+09,9E+09,9E+09,9E+09,9E+09,9E+09]];
	CONST robtarget Target_2960:=[[402.8,-204.2,-122],[-0.0726551899005905,-0.464469513168276,0.870394556627551,0.146296310653628],[0,0,0,1],[9E+09,9E+09,9E+09,9E+09,9E+09,9E+09]];
	CONST robtarget Target_2970:=[[402.8,-199.5,-121.1],[-0.0732513409768337,-0.467177259971663,0.86918784700694,0.144541120190431],[0,0,0,1],[9E+09,9E+09,9E+09,9E+09,9E+09,9E+09]];
	CONST robtarget Target_2980:=[[402.8,-194.7,-120.2],[-0.0738556750281974,-0.469888165079486,0.867963924187749,0.142790328429366],[0,0,0,1],[9E+09,9E+09,9E+09,9E+09,9E+09,9E+09]];
	CONST robtarget Target_2990:=[[402.8,-190,-119.4],[-0.0744838693064031,-0.47250573765079,0.866775279580614,0.141035796194364],[0,0,0,1],[9E+09,9E+09,9E+09,9E+09,9E+09,9E+09]];
	CONST robtarget Target_3000:=[[402.8,-185.2,-118.6],[-0.0751271551758748,-0.475123352543578,0.865568767967733,0.139299742791405],[0,0,0,1],[9E+09,9E+09,9E+09,9E+09,9E+09,9E+09]];
	CONST robtarget Target_3010:=[[402.8,-180.5,-117.8],[-0.0757931074196912,-0.477651409177404,0.864396792123501,0.137559884941466],[0,0,0,1],[9E+09,9E+09,9E+09,9E+09,9E+09,9E+09]];
	CONST robtarget Target_3020:=[[402.8,-175.7,-117],[-0.0764665486570193,-0.480183058736185,0.863208454893834,0.135824373508752],[0,0,0,1],[9E+09,9E+09,9E+09,9E+09,9E+09,9E+09]];
	CONST robtarget Target_3030:=[[402.8,-171,-116.2],[-0.0771614116925029,-0.482628601670918,0.862053869763887,0.134085327384847],[0,0,0,1],[9E+09,9E+09,9E+09,9E+09,9E+09,9E+09]];
	CONST robtarget Target_3040:=[[402.8,-166.2,-115.5],[-0.0778709701289027,-0.485074868994747,0.860882254846597,0.132363993484447],[0,0,0,1],[9E+09,9E+09,9E+09,9E+09,9E+09,9E+09]];
	CONST robtarget Target_3050:=[[402.8,-161.5,-114.7],[-0.0785932462996557,-0.487441371392645,0.859744651172031,0.130625977018442],[0,0,0,1],[9E+09,9E+09,9E+09,9E+09,9E+09,9E+09]];
	CONST robtarget Target_3060:=[[402.8,-156.7,-114],[-0.0793299911579505,-0.48980884043689,0.858590377213851,0.128905455619714],[0,0,0,1],[9E+09,9E+09,9E+09,9E+09,9E+09,9E+09]];
	CONST robtarget Target_3070:=[[402.8,-152,-113.4],[-0.0800859892650813,-0.492096745025681,0.85746829812881,0.127181545684289],[0,0,0,1],[9E+09,9E+09,9E+09,9E+09,9E+09,9E+09]];
	CONST robtarget Target_3080:=[[402.8,-147.2,-112.7],[-0.0808485209568348,-0.494388693142767,0.85633090303092,0.125462031172498],[0,0,0,1],[9E+09,9E+09,9E+09,9E+09,9E+09,9E+09]];
	CONST robtarget Target_3090:=[[402.8,-142.5,-112.1],[-0.0816371898293487,-0.496601394139729,0.855223911280943,0.123751711699554],[0,0,0,1],[9E+09,9E+09,9E+09,9E+09,9E+09,9E+09]];
	CONST robtarget Target_3100:=[[402.8,-137.7,-111.5],[-0.0824241810789566,-0.498820929796159,0.854102914285517,0.122033381415685],[0,0,0,1],[9E+09,9E+09,9E+09,9E+09,9E+09,9E+09]];
	CONST robtarget Target_3110:=[[402.8,-133,-110.9],[-0.0832364492410585,-0.500964173166576,0.853011546080285,0.120324116348267],[0,0,0,1],[9E+09,9E+09,9E+09,9E+09,9E+09,9E+09]];
	CONST robtarget Target_3120:=[[402.8,-128.2,-110.3],[-0.0840547505157918,-0.503111723230313,0.851905448022469,0.118619140502658],[0,0,0,1],[9E+09,9E+09,9E+09,9E+09,9E+09,9E+09]];
	CONST robtarget Target_3130:=[[402.8,-123.5,-109.7],[-0.0848894135021422,-0.505188317055692,0.850829213294253,0.116911084122863],[0,0,0,1],[9E+09,9E+09,9E+09,9E+09,9E+09,9E+09]];
	CONST robtarget Target_3140:=[[402.8,-118.7,-109.2],[-0.0857298016167959,-0.507269262415874,0.849738515063917,0.115207432658531],[0,0,0,1],[9E+09,9E+09,9E+09,9E+09,9E+09,9E+09]];
	CONST robtarget Target_3150:=[[402.8,-114,-108.7],[-0.086594071211112,-0.509279539964095,0.848675906562912,0.113512213548427],[0,0,0,1],[9E+09,9E+09,9E+09,9E+09,9E+09,9E+09]];
	CONST robtarget Target_3160:=[[402.8,-109.2,-108.2],[-0.0874639394061394,-0.511294325848003,0.847599078876557,0.111821165915971],[0,0,0,1],[9E+09,9E+09,9E+09,9E+09,9E+09,9E+09]];
	CONST robtarget Target_3170:=[[402.8,-104.5,-107.7],[-0.0883399330737308,-0.513245410221675,0.846551620286965,0.110116117350853],[0,0,0,1],[9E+09,9E+09,9E+09,9E+09,9E+09,9E+09]];
	CONST robtarget Target_3180:=[[402.8,-99.7,-107.3],[-0.0892384702830976,-0.515196733091968,0.845488129365696,0.108437284799062],[0,0,0,1],[9E+09,9E+09,9E+09,9E+09,9E+09,9E+09]];
	CONST robtarget Target_3190:=[[402.8,-95,-106.9],[-0.0901423003837138,-0.517086668114792,0.844453270290143,0.106744637503524],[0,0,0,1],[9E+09,9E+09,9E+09,9E+09,9E+09,9E+09]];
	CONST robtarget Target_3200:=[[402.8,-90.2,-106.5],[-0.0910511707405547,-0.518981138934832,0.843404658938233,0.10505638018684],[0,0,0,1],[9E+09,9E+09,9E+09,9E+09,9E+09,9E+09]];
	CONST robtarget Target_3210:=[[402.8,-85.5,-106.1],[-0.0919821292202773,-0.520812375289864,0.842381870286688,0.103375733425865],[0,0,0,1],[9E+09,9E+09,9E+09,9E+09,9E+09,9E+09]];
	CONST robtarget Target_3220:=[[402.8,-80.7,-105.7],[-0.0929180477631145,-0.522648262706537,0.841345526352199,0.101699238821492],[0,0,0,1],[9E+09,9E+09,9E+09,9E+09,9E+09,9E+09]];
	CONST robtarget Target_3230:=[[402.8,-76,-105.4],[-0.0938665059487625,-0.524425036468661,0.84033533676462,0.10001990787092],[0,0,0,1],[9E+09,9E+09,9E+09,9E+09,9E+09,9E+09]];
	CONST robtarget Target_3240:=[[402.8,-71.2,-105.1],[-0.0948196695426027,-0.526206448577127,0.839311799840147,0.0983448340929584],[0,0,0,1],[9E+09,9E+09,9E+09,9E+09,9E+09,9E+09]];
	CONST robtarget Target_3250:=[[402.8,-66.5,-104.8],[-0.0957846493359272,-0.527930745779311,0.838313724949949,0.0966670945722251],[0,0,0,1],[9E+09,9E+09,9E+09,9E+09,9E+09,9E+09]];
	CONST robtarget Target_3260:=[[402.8,-61.7,-104.5],[-0.0967635456695024,-0.529658037088889,0.837301369836592,0.0950031370344002],[0,0,0,1],[9E+09,9E+09,9E+09,9E+09,9E+09,9E+09]];
	CONST robtarget Target_3270:=[[402.8,-57,-104.2],[-0.0977442049376423,-0.531331798074137,0.836314920035596,0.0933270876126915],[0,0,0,1],[9E+09,9E+09,9E+09,9E+09,9E+09,9E+09]];
	CONST robtarget Target_3280:=[[402.8,-52.2,-104],[-0.0987387394706192,-0.533008633679001,0.835314349416395,0.0916645810030375],[0,0,0,1],[9E+09,9E+09,9E+09,9E+09,9E+09,9E+09]];
	CONST robtarget Target_3290:=[[402.8,-47.5,-103.8],[-0.0997439357155413,-0.53463218512944,0.834337870776175,0.0899993961111565],[0,0,0,1],[9E+09,9E+09,9E+09,9E+09,9E+09,9E+09]];
	CONST robtarget Target_3300:=[[402.8,-42.7,-103.6],[-0.100763181264532,-0.536258987956148,0.833347380044937,0.0883471748837484],[0,0,0,1],[9E+09,9E+09,9E+09,9E+09,9E+09,9E+09]];
	CONST robtarget Target_3310:=[[402.8,-38,-103.4],[-0.101782695272046,-0.537835700102673,0.832381528602919,0.0866835248411941],[0,0,0,1],[9E+09,9E+09,9E+09,9E+09,9E+09,9E+09]];
	CONST robtarget Target_3320:=[[402.8,-33.2,-103.2],[-0.102816242063543,-0.539415722987032,0.83140180114988,0.0850326008483989],[0,0,0,1],[9E+09,9E+09,9E+09,9E+09,9E+09,9E+09]];
	CONST robtarget Target_3330:=[[402.8,-28.5,-103.1],[-0.103849243809564,-0.540947203735296,0.830446130899949,0.0833707442958957],[0,0,0,1],[9E+09,9E+09,9E+09,9E+09,9E+09,9E+09]];
	CONST robtarget Target_3340:=[[402.8,-23.7,-103],[-0.104896269655517,-0.542482047153467,0.829476713310843,0.0817213754386389],[0,0,0,1],[9E+09,9E+09,9E+09,9E+09,9E+09,9E+09]];
	CONST robtarget Target_3350:=[[402.8,-19,-102.9],[-0.105962742127289,-0.543967513189088,0.828528128312723,0.0800773530429236],[0,0,0,1],[9E+09,9E+09,9E+09,9E+09,9E+09,9E+09]];
	CONST robtarget Target_3360:=[[402.8,-14.2,-102.8],[-0.107022669132324,-0.545458796532891,0.827568528802926,0.0784294569128447],[0,0,0,1],[9E+09,9E+09,9E+09,9E+09,9E+09,9E+09]];
	CONST robtarget Target_3370:=[[402.8,-9.5,-102.8],[-0.108091093958442,-0.546903363962133,0.826630501210307,0.0767791662013001],[0,0,0,1],[9E+09,9E+09,9E+09,9E+09,9E+09,9E+09]];
	CONST robtarget Target_3380:=[[402.8,-4.7,-102.7],[-0.109173771339137,-0.548351470788281,0.82567890219086,0.0751405523856116],[0,0,0,1],[9E+09,9E+09,9E+09,9E+09,9E+09,9E+09]];
	CONST robtarget Target_3390:=[[402.8,0,-102.7],[-0.110264632104129,-0.549754394983045,0.824748240673187,0.0734993578900568],[0,0,0,1],[9E+09,9E+09,9E+09,9E+09,9E+09,9E+09]];
	CONST robtarget Target_3400:=[[407.4,0,-104],[-0.110504668218722,-0.547051333715954,0.826543642874522,0.0731379723890373],[0,0,0,1],[9E+09,9E+09,9E+09,9E+09,9E+09,9E+09]];
	CONST robtarget Target_3410:=[[412.2,0,-105.3],[-0.110752473630896,-0.544240484714039,0.828397157222862,0.0727621762177796],[0,0,0,1],[9E+09,9E+09,9E+09,9E+09,9E+09,9E+09]];
	CONST robtarget Target_3420:=[[416.9,0,-106.6],[-0.11099248585662,-0.541498075946965,0.830192380742214,0.0723955301567542],[0,0,0,1],[9E+09,9E+09,9E+09,9E+09,9E+09,9E+09]];
	CONST robtarget Target_3430:=[[421.6,0,-107.9],[-0.111229904640411,-0.538765681366938,0.831968206049912,0.0720302229414467],[0,0,0,1],[9E+09,9E+09,9E+09,9E+09,9E+09,9E+09]];
	CONST robtarget Target_3440:=[[426.3,0,-109.1],[-0.111464740101592,-0.536043529178033,0.833724708835626,0.071666285081578],[0,0,0,1],[9E+09,9E+09,9E+09,9E+09,9E+09,9E+09]];
	CONST robtarget Target_3450:=[[431,0,-110.4],[-0.111697003073208,-0.533331840196533,0.835461970127468,0.0713037460991586],[0,0,0,1],[9E+09,9E+09,9E+09,9E+09,9E+09,9E+09]];
	CONST robtarget Target_3460:=[[435.7,0,-111.7],[-0.11192670507555,-0.530630827871887,0.837180076093959,0.0709426345312907],[0,0,0,1],[9E+09,9E+09,9E+09,9E+09,9E+09,9E+09]];
	CONST robtarget Target_3470:=[[440.5,0,-113],[-0.112158663737912,-0.527883581221801,0.838915061238703,0.0705753416699882],[0,0,0,1],[9E+09,9E+09,9E+09,9E+09,9E+09,9E+09]];
	CONST robtarget Target_3480:=[[445.2,0,-114.3],[-0.112383227166656,-0.525204771126114,0.840594732129019,0.0702171984268614],[0,0,0,1],[9E+09,9E+09,9E+09,9E+09,9E+09,9E+09]];
	CONST robtarget Target_3490:=[[449.9,0,-115.6],[-0.11260526833937,-0.522537238151298,0.842255537258084,0.069860562877262],[0,0,0,1],[9E+09,9E+09,9E+09,9E+09,9E+09,9E+09]];
	CONST robtarget Target_3500:=[[454.6,0,-116.8],[-0.112824801275096,-0.519881166480892,0.843897581484363,0.0695054596455891],[0,0,0,1],[9E+09,9E+09,9E+09,9E+09,9E+09,9E+09]];
	CONST robtarget Target_3510:=[[459.3,0,-118.1],[-0.113041840549329,-0.517236733143435,0.845520973828442,0.0691519123996556],[0,0,0,1],[9E+09,9E+09,9E+09,9E+09,9E+09,9E+09]];
	CONST robtarget Target_3520:=[[464.1,0,-119.4],[-0.113260939575128,-0.514548224271978,0.847159772531277,0.0687924724796892],[0,0,0,1],[9E+09,9E+09,9E+09,9E+09,9E+09,9E+09]];
	CONST robtarget Target_3530:=[[468.8,0,-120.7],[-0.113472985122302,-0.511927826802447,0.848745813210301,0.0684421387066719],[0,0,0,1],[9E+09,9E+09,9E+09,9E+09,9E+09,9E+09]];
	CONST robtarget Target_3540:=[[473.5,0,-122],[-0.113682584168509,-0.509319559704371,0.850313554754501,0.0680934267024318],[0,0,0,1],[9E+09,9E+09,9E+09,9E+09,9E+09,9E+09]];
	CONST robtarget Target_3550:=[[478.2,0,-123.3],[-0.11388975327396,-0.506723571907233,0.851863121029585,0.067746356378081],[0,0,0,1],[9E+09,9E+09,9E+09,9E+09,9E+09,9E+09]];
	CONST robtarget Target_3560:=[[482.9,0,-124.5],[-0.11409450943123,-0.504140005546083,0.853394639135193,0.0674009467363505],[0,0,0,1],[9E+09,9E+09,9E+09,9E+09,9E+09,9E+09]];
	CONST robtarget Target_3570:=[[487.6,0,-125.8],[-0.114296870041643,-0.501568996047657,0.854908239228302,0.0670572158831039],[0,0,0,1],[9E+09,9E+09,9E+09,9E+09,9E+09,9E+09]];
	CONST robtarget Target_3580:=[[492.4,0,-127.1],[-0.114501082145061,-0.49895637853071,0.856435687965074,0.0667079222500556],[0,0,0,1],[9E+09,9E+09,9E+09,9E+09,9E+09,9E+09]];
	CONST robtarget Target_3590:=[[497.1,0,-128.4],[-0.114698655380453,-0.496411136450267,0.857913479847965,0.066367636369134],[0,0,0,1],[9E+09,9E+09,9E+09,9E+09,9E+09,9E+09]];
	CONST robtarget Target_3600:=[[497.1,-4.8,-128.4],[-0.113685772876722,-0.494647900083909,0.858928398856533,0.0681249266109921],[0,0,0,1],[9E+09,9E+09,9E+09,9E+09,9E+09,9E+09]];
	CONST robtarget Target_3610:=[[497.1,-9.7,-128.5],[-0.112719580475348,-0.492834933972254,0.859959428792142,0.0698412833896862],[0,0,0,1],[9E+09,9E+09,9E+09,9E+09,9E+09,9E+09]];
	CONST robtarget Target_3620:=[[497.1,-14.5,-128.5],[-0.111721708687057,-0.491025084092936,0.860979678217218,0.0716004210640201],[0,0,0,1],[9E+09,9E+09,9E+09,9E+09,9E+09,9E+09]];
	CONST robtarget Target_3630:=[[497.1,-19.3,-128.6],[-0.110742542845466,-0.489190564236867,0.862001094207298,0.0733675313143067],[0,0,0,1],[9E+09,9E+09,9E+09,9E+09,9E+09,9E+09]];
	CONST robtarget Target_3640:=[[497.1,-24.1,-128.7],[-0.109796606270312,-0.487338272515718,0.863022277739868,0.0750910215512359],[0,0,0,1],[9E+09,9E+09,9E+09,9E+09,9E+09,9E+09]];
	CONST robtarget Target_3650:=[[497.1,-29,-128.8],[-0.108836261807873,-0.485421741269383,0.864068044924914,0.076855806275945],[0,0,0,1],[9E+09,9E+09,9E+09,9E+09,9E+09,9E+09]];
	CONST robtarget Target_3660:=[[497.1,-33.8,-128.9],[-0.107881292685985,-0.483513693138095,0.865097763106697,0.0786256669551985],[0,0,0,1],[9E+09,9E+09,9E+09,9E+09,9E+09,9E+09]];
	CONST robtarget Target_3670:=[[497.1,-38.6,-129.1],[-0.106934802533463,-0.481580560229526,0.866130214185355,0.0803962940151815],[0,0,0,1],[9E+09,9E+09,9E+09,9E+09,9E+09,9E+09]];
	CONST robtarget Target_3680:=[[497.1,-43.4,-129.3],[-0.106032467084069,-0.47962714228744,0.86716170499343,0.0821309789186549],[0,0,0,1],[9E+09,9E+09,9E+09,9E+09,9E+09,9E+09]];
	CONST robtarget Target_3690:=[[497.1,-48.3,-129.5],[-0.105117139403384,-0.477605783216225,0.868218123595881,0.0839070479859285],[0,0,0,1],[9E+09,9E+09,9E+09,9E+09,9E+09,9E+09]];
	CONST robtarget Target_3700:=[[497.1,-53.1,-129.7],[-0.104207441869202,-0.47559319696472,0.869257981542432,0.0856882814901278],[0,0,0,1],[9E+09,9E+09,9E+09,9E+09,9E+09,9E+09]];
	CONST robtarget Target_3710:=[[497.1,-57.9,-130],[-0.103306925600619,-0.473553916791643,0.870300702751293,0.0874703024165777],[0,0,0,1],[9E+09,9E+09,9E+09,9E+09,9E+09,9E+09]];
	CONST robtarget Target_3720:=[[497.1,-62.8,-130.3],[-0.102454384453759,-0.471455636967711,0.871363176577917,0.0892126447406036],[0,0,0,1],[9E+09,9E+09,9E+09,9E+09,9E+09,9E+09]];
	CONST robtarget Target_3730:=[[497.1,-67.6,-130.6],[-0.101582810653362,-0.4693596378167,0.872410754293778,0.0910051578807516],[0,0,0,1],[9E+09,9E+09,9E+09,9E+09,9E+09,9E+09]];
	CONST robtarget Target_3740:=[[497.1,-72.4,-130.9],[-0.100711100593576,-0.467237315650497,0.873462480482747,0.0927893327375243],[0,0,0,1],[9E+09,9E+09,9E+09,9E+09,9E+09,9E+09]];
	CONST robtarget Target_3750:=[[497.1,-77.2,-131.2],[-0.0998935205336521,-0.46509010451507,0.874513118442847,0.094547791666017],[0,0,0,1],[9E+09,9E+09,9E+09,9E+09,9E+09,9E+09]];
	CONST robtarget Target_3760:=[[497.1,-82.1,-131.6],[-0.099056043463908,-0.462869629811393,0.875590401674392,0.0963382299360835],[0,0,0,1],[9E+09,9E+09,9E+09,9E+09,9E+09,9E+09]];
	CONST robtarget Target_3770:=[[497.1,-86.9,-132],[-0.0982248398131066,-0.460658557283113,0.876650073487825,0.0981337001204021],[0,0,0,1],[9E+09,9E+09,9E+09,9E+09,9E+09,9E+09]];
	CONST robtarget Target_3780:=[[497.1,-91.7,-132.4],[-0.0974138642079185,-0.458415825254638,0.877711534519642,0.0999396437224223],[0,0,0,1],[9E+09,9E+09,9E+09,9E+09,9E+09,9E+09]];
	CONST robtarget Target_3790:=[[497.1,-96.5,-132.8],[-0.0966377890242803,-0.456149949094279,0.878774831163567,0.101701316546196],[0,0,0,1],[9E+09,9E+09,9E+09,9E+09,9E+09,9E+09]];
	CONST robtarget Target_3800:=[[497.1,-101.4,-133.2],[-0.0958534839166685,-0.453804683861292,0.879863796394934,0.103504194698011],[0,0,0,1],[9E+09,9E+09,9E+09,9E+09,9E+09,9E+09]];
	CONST robtarget Target_3810:=[[497.1,-106.2,-133.7],[-0.0950757836771643,-0.451469158033298,0.880934470350742,0.105312172376874],[0,0,0,1],[9E+09,9E+09,9E+09,9E+09,9E+09,9E+09]];
	CONST robtarget Target_3820:=[[497.1,-111,-134.2],[-0.0943426941848549,-0.449107069461519,0.882006145432098,0.107086206551745],[0,0,0,1],[9E+09,9E+09,9E+09,9E+09,9E+09,9E+09]];
	CONST robtarget Target_3830:=[[497.1,-115.8,-134.7],[-0.0935883247365094,-0.446707677832054,0.883082840198059,0.108895240422325],[0,0,0,1],[9E+09,9E+09,9E+09,9E+09,9E+09,9E+09]];
	CONST robtarget Target_3840:=[[497.1,-120.7,-135.3],[-0.0928607089574246,-0.444229292117783,0.884183408461757,0.110710997454669],[0,0,0,1],[9E+09,9E+09,9E+09,9E+09,9E+09,9E+09]];
	CONST robtarget Target_3850:=[[497.1,-125.5,-135.8],[-0.09216351759295,-0.441768481872784,0.885264498048338,0.112486723411854],[0,0,0,1],[9E+09,9E+09,9E+09,9E+09,9E+09,9E+09]];
	CONST robtarget Target_3860:=[[497.1,-130.3,-136.4],[-0.0914643039208925,-0.439264011055841,0.886347823416698,0.114319489256572],[0,0,0,1],[9E+09,9E+09,9E+09,9E+09,9E+09,9E+09]];
	CONST robtarget Target_3870:=[[497.1,-135.2,-137],[-0.0907750220715357,-0.436681615636182,0.887457795723534,0.116136655465931],[0,0,0,1],[9E+09,9E+09,9E+09,9E+09,9E+09,9E+09]];
	CONST robtarget Target_3880:=[[497.1,-140,-137.6],[-0.0901019068934567,-0.434107137934023,0.888546900758733,0.117970523101938],[0,0,0,1],[9E+09,9E+09,9E+09,9E+09,9E+09,9E+09]];
	CONST robtarget Target_3890:=[[497.1,-144.8,-138.3],[-0.089465176247308,-0.431504836817279,0.889638798139368,0.119759621273083],[0,0,0,1],[9E+09,9E+09,9E+09,9E+09,9E+09,9E+09]];
	CONST robtarget Target_3900:=[[497.1,-149.6,-139],[-0.0888190416506828,-0.428858874632301,0.890733439707747,0.121594337350781],[0,0,0,1],[9E+09,9E+09,9E+09,9E+09,9E+09,9E+09]];
	CONST robtarget Target_3910:=[[497.1,-154.5,-139.7],[-0.0881936860705587,-0.426127526136662,0.891854024804215,0.123424485603378],[0,0,0,1],[9E+09,9E+09,9E+09,9E+09,9E+09,9E+09]];
	CONST robtarget Target_3920:=[[497.1,-159.3,-140.4],[-0.0875846747965808,-0.423404259194089,0.892952775543361,0.12527209859538],[0,0,0,1],[9E+09,9E+09,9E+09,9E+09,9E+09,9E+09]];
	CONST robtarget Target_3930:=[[497.1,-164.1,-141.1],[-0.0870042211294205,-0.420653943782027,0.894055790207633,0.127062067834958],[0,0,0,1],[9E+09,9E+09,9E+09,9E+09,9E+09,9E+09]];
	CONST robtarget Target_3940:=[[497.1,-169,-141.9],[-0.0864319560074965,-0.417803485327623,0.895183340350478,0.128905204657413],[0,0,0,1],[9E+09,9E+09,9E+09,9E+09,9E+09,9E+09]];
	CONST robtarget Target_3950:=[[497.1,-173.8,-142.7],[-0.0858677901272042,-0.414964306568703,0.896289519475067,0.130753371550333],[0,0,0,1],[9E+09,9E+09,9E+09,9E+09,9E+09,9E+09]];
	CONST robtarget Target_3960:=[[497.1,-178.6,-143.5],[-0.0853496583053356,-0.412090385819937,0.897397507883673,0.132569463248934],[0,0,0,1],[9E+09,9E+09,9E+09,9E+09,9E+09,9E+09]];
	CONST robtarget Target_3970:=[[497.1,-183.4,-144.3],[-0.0848168422216677,-0.409171395039952,0.898508073561403,0.134417686714142],[0,0,0,1],[9E+09,9E+09,9E+09,9E+09,9E+09,9E+09]];
	CONST robtarget Target_3980:=[[497.1,-188.3,-145.2],[-0.0843167878090531,-0.406154114139921,0.899643737945273,0.136274207525252],[0,0,0,1],[9E+09,9E+09,9E+09,9E+09,9E+09,9E+09]];
	CONST robtarget Target_3990:=[[497.1,-193.1,-146.1],[-0.0838469974622208,-0.403156804975992,0.90075819436766,0.138090357728671],[0,0,0,1],[9E+09,9E+09,9E+09,9E+09,9E+09,9E+09]];
	CONST robtarget Target_4000:=[[497.1,-197.9,-147],[-0.0833723294284235,-0.400109234116158,0.901873147936863,0.139951707710602],[0,0,0,1],[9E+09,9E+09,9E+09,9E+09,9E+09,9E+09]];
	CONST robtarget Target_4010:=[[497.1,-202.7,-147.9],[-0.0829149781121735,-0.397018868118146,0.902989630044964,0.141812738476147],[0,0,0,1],[9E+09,9E+09,9E+09,9E+09,9E+09,9E+09]];
	CONST robtarget Target_4020:=[[497.1,-207.6,-148.8],[-0.0824925655481992,-0.393823892416875,0.904131118195996,0.143682425858401],[0,0,0,1],[9E+09,9E+09,9E+09,9E+09,9E+09,9E+09]];
	CONST robtarget Target_4030:=[[497.1,-212.4,-149.8],[-0.0821003495685957,-0.390649711482271,0.905250623606648,0.145511662691714],[0,0,0,1],[9E+09,9E+09,9E+09,9E+09,9E+09,9E+09]];
	CONST robtarget Target_4040:=[[497.1,-217.2,-150.8],[-0.0817052988122214,-0.387422415146083,0.906369414376248,0.14738589169808],[0,0,0,1],[9E+09,9E+09,9E+09,9E+09,9E+09,9E+09]];
	CONST robtarget Target_4050:=[[497.1,-222,-151.8],[-0.0813290537624266,-0.384149608847722,0.907488980773307,0.149259548476051],[0,0,0,1],[9E+09,9E+09,9E+09,9E+09,9E+09,9E+09]];
	CONST robtarget Target_4060:=[[497.1,-226.9,-152.8],[-0.0810028238309002,-0.380777830631852,0.908636966983253,0.151081595378776],[0,0,0,1],[9E+09,9E+09,9E+09,9E+09,9E+09,9E+09]];
	CONST robtarget Target_4070:=[[501.8,-226.6,-154.1],[-0.081484535312662,-0.377876295599331,0.909847459354232,0.150822334008115],[0,0,0,1],[9E+09,9E+09,9E+09,9E+09,9E+09,9E+09]];
	CONST robtarget Target_4080:=[[506.5,-226.3,-155.3],[-0.0819589608488699,-0.375009977883674,0.911032606747371,0.15056505128133],[0,0,0,1],[9E+09,9E+09,9E+09,9E+09,9E+09,9E+09]];
	CONST robtarget Target_4090:=[[511.2,-226,-156.6],[-0.0824262210994575,-0.3721784984148,0.912192994594307,0.15030976018223],[0,0,0,1],[9E+09,9E+09,9E+09,9E+09,9E+09,9E+09]];
	CONST robtarget Target_4100:=[[515.9,-225.7,-157.8],[-0.0828864355388679,-0.369381474041948,0.913329196239681,0.150056471817903],[0,0,0,1],[9E+09,9E+09,9E+09,9E+09,9E+09,9E+09]];
	CONST robtarget Target_4110:=[[520.6,-225.4,-159.1],[-0.0833397223953481,-0.366618518161673,0.91444177300152,0.149805195510177],[0,0,0,1],[9E+09,9E+09,9E+09,9E+09,9E+09,9E+09]];
	CONST robtarget Target_4120:=[[525.4,-225.1,-160.3],[-0.0838160442684706,-0.363835960211449,0.915558118343285,0.149504503998719],[0,0,0,1],[9E+09,9E+09,9E+09,9E+09,9E+09,9E+09]];
	CONST robtarget Target_4130:=[[530.1,-224.8,-161.6],[-0.0842555477574826,-0.36114066646297,0.916624619478424,0.149257256657101],[0,0,0,1],[9E+09,9E+09,9E+09,9E+09,9E+09,9E+09]];
	CONST robtarget Target_4140:=[[534.8,-224.5,-162.8],[-0.084688474326446,-0.358478258694518,0.917669119045982,0.149012040818775],[0,0,0,1],[9E+09,9E+09,9E+09,9E+09,9E+09,9E+09]];
	CONST robtarget Target_4150:=[[539.5,-224.2,-164.1],[-0.0851149366853577,-0.355848342035156,0.918692130954714,0.148768859462472],[0,0,0,1],[9E+09,9E+09,9E+09,9E+09,9E+09,9E+09]];
	CONST robtarget Target_4160:=[[544.2,-224,-165.3],[-0.0855449919953143,-0.353188933010917,0.919717810856076,0.148521986039909],[0,0,0,1],[9E+09,9E+09,9E+09,9E+09,9E+09,9E+09]];
	CONST robtarget Target_4170:=[[548.9,-223.6,-166.6],[-0.0859680323867778,-0.350692718960615,0.920678155733562,0.148242530437806],[0,0,0,1],[9E+09,9E+09,9E+09,9E+09,9E+09,9E+09]];
	CONST robtarget Target_4180:=[[553.7,-223.4,-167.8],[-0.0863947561666026,-0.348038828247146,0.921684666037846,0.147994244921791],[0,0,0,1],[9E+09,9E+09,9E+09,9E+09,9E+09,9E+09]];
	CONST robtarget Target_4190:=[[558.4,-223.1,-169.1],[-0.0867961732530741,-0.345535601674814,0.922626033424251,0.147759178163931],[0,0,0,1],[9E+09,9E+09,9E+09,9E+09,9E+09,9E+09]];
	CONST robtarget Target_4200:=[[563.1,-222.8,-170.3],[-0.0871916700771293,-0.34306288786098,0.92354832280148,0.147526143758382],[0,0,0,1],[9E+09,9E+09,9E+09,9E+09,9E+09,9E+09]];
	CONST robtarget Target_4210:=[[567.8,-222.5,-171.6],[-0.0875813502222025,-0.340620292727912,0.9244519813159,0.147295137449658],[0,0,0,1],[9E+09,9E+09,9E+09,9E+09,9E+09,9E+09]];
	CONST robtarget Target_4220:=[[572.5,-222.2,-172.8],[-0.0879838114415392,-0.338215709016228,0.925340021263495,0.14701982229259],[0,0,0,1],[9E+09,9E+09,9E+09,9E+09,9E+09,9E+09]];
	CONST robtarget Target_4230:=[[577.2,-221.9,-174.1],[-0.0883620433130744,-0.335832168276347,0.92620773886212,0.146792808148981],[0,0,0,1],[9E+09,9E+09,9E+09,9E+09,9E+09,9E+09]];
	CONST robtarget Target_4240:=[[582,-221.6,-175.3],[-0.0887432500085563,-0.333423879444064,0.927077417152281,0.146562665098053],[0,0,0,1],[9E+09,9E+09,9E+09,9E+09,9E+09,9E+09]];
	CONST robtarget Target_4250:=[[586.7,-221.3,-176.6],[-0.0891104346648562,-0.331098452423926,0.927910467437326,0.146339706356701],[0,0,0,1],[9E+09,9E+09,9E+09,9E+09,9E+09,9E+09]];
	CONST robtarget Target_4260:=[[492.4,-227.2,-151.6],[-0.0804929335251649,-0.383706552397799,0.907398364231878,0.151388169580122],[0,0,0,1],[9E+09,9E+09,9E+09,9E+09,9E+09,9E+09]];
	CONST robtarget Target_4270:=[[487.6,-227.5,-150.3],[-0.0799848305294338,-0.386747176931651,0.906106578112692,0.15165723563841],[0,0,0,1],[9E+09,9E+09,9E+09,9E+09,9E+09,9E+09]];
	CONST robtarget Target_4280:=[[482.9,-227.8,-149.1],[-0.079480211101064,-0.389757348968478,0.904815847942971,0.151922303430526],[0,0,0,1],[9E+09,9E+09,9E+09,9E+09,9E+09,9E+09]];
	CONST robtarget Target_4290:=[[478.2,-228.1,-147.8],[-0.0789755718638235,-0.392800282298334,0.903495759273722,0.152204501410216],[0,0,0,1],[9E+09,9E+09,9E+09,9E+09,9E+09,9E+09]];
	CONST robtarget Target_4300:=[[473.5,-228.3,-146.6],[-0.0784449698780569,-0.395944743888569,0.902122169435086,0.152478647362774],[0,0,0,1],[9E+09,9E+09,9E+09,9E+09,9E+09,9E+09]];
	CONST robtarget Target_4310:=[[468.8,-228.7,-145.3],[-0.0779052718552005,-0.39899698285581,0.900770595559414,0.152789104535194],[0,0,0,1],[9E+09,9E+09,9E+09,9E+09,9E+09,9E+09]];
	CONST robtarget Target_4320:=[[464.1,-228.9,-144.1],[-0.0773583028575654,-0.402216157514004,0.899337767908794,0.153066765911142],[0,0,0,1],[9E+09,9E+09,9E+09,9E+09,9E+09,9E+09]];
	CONST robtarget Target_4330:=[[459.3,-229.2,-142.8],[-0.0768009502507997,-0.405485191721261,0.897868596982472,0.153347174372641],[0,0,0,1],[9E+09,9E+09,9E+09,9E+09,9E+09,9E+09]];
	CONST robtarget Target_4340:=[[454.6,-229.5,-141.6],[-0.0762473421058434,-0.40872108006576,0.8964002102088,0.153623190532203],[0,0,0,1],[9E+09,9E+09,9E+09,9E+09,9E+09,9E+09]];
	CONST robtarget Target_4350:=[[449.9,-229.8,-140.3],[-0.0756851876260789,-0.411995579065772,0.894899939089706,0.15390092339393],[0,0,0,1],[9E+09,9E+09,9E+09,9E+09,9E+09,9E+09]];
	CONST robtarget Target_4360:=[[445.2,-230.1,-139.1],[-0.0751143593956152,-0.415308968869869,0.893367068191316,0.154180332273884],[0,0,0,1],[9E+09,9E+09,9E+09,9E+09,9E+09,9E+09]];
	CONST robtarget Target_4370:=[[440.5,-230.4,-137.8],[-0.0745122120906639,-0.418653028889783,0.891799026990306,0.154505880502683],[0,0,0,1],[9E+09,9E+09,9E+09,9E+09,9E+09,9E+09]];
	CONST robtarget Target_4380:=[[435.7,-230.7,-136.6],[-0.0739102097740581,-0.42212132118016,0.890162599385395,0.154794760091252],[0,0,0,1],[9E+09,9E+09,9E+09,9E+09,9E+09,9E+09]];
	CONST robtarget Target_4390:=[[431,-231,-135.3],[-0.0733122343663245,-0.425553728621472,0.888526807246585,0.155078861076456],[0,0,0,1],[9E+09,9E+09,9E+09,9E+09,9E+09,9E+09]];
	CONST robtarget Target_4400:=[[426.3,-231.3,-134.1],[-0.0727050748938696,-0.429025989563119,0.886855435467829,0.155364439126946],[0,0,0,1],[9E+09,9E+09,9E+09,9E+09,9E+09,9E+09]];
	CONST robtarget Target_4410:=[[421.6,-231.6,-132.8],[-0.0720886068461626,-0.432538296849065,0.885147719252757,0.155651436304112],[0,0,0,1],[9E+09,9E+09,9E+09,9E+09,9E+09,9E+09]];
	CONST robtarget Target_4420:=[[416.9,-231.9,-131.6],[-0.0714627069387675,-0.436090821962743,0.883402885516742,0.155939790873072],[0,0,0,1],[9E+09,9E+09,9E+09,9E+09,9E+09,9E+09]];
	CONST robtarget Target_4430:=[[412.2,-232.2,-130.3],[-0.0708036869949546,-0.439675185640343,0.881618508706087,0.156273395518577],[0,0,0,1],[9E+09,9E+09,9E+09,9E+09,9E+09,9E+09]];
	CONST robtarget Target_4440:=[[407.4,-232.5,-129.1],[-0.0701438997920973,-0.443389919698404,0.879756126929991,0.156570653575124],[0,0,0,1],[9E+09,9E+09,9E+09,9E+09,9E+09,9E+09]];
	CONST robtarget Target_4450:=[[303.7,-238.9,-101.6],[-0.0531406589164049,-0.533770858467849,0.828019948764244,0.16324124928732],[0,0,0,1],[9E+09,9E+09,9E+09,9E+09,9E+09,9E+09]];
	CONST robtarget Target_4460:=[[299,-239.2,-100.3],[-0.0522188939240138,-0.538281296648858,0.82508859631501,0.163570293838167],[0,0,0,1],[9E+09,9E+09,9E+09,9E+09,9E+09,9E+09]];
	CONST robtarget Target_4470:=[[294.2,-239.5,-99.1],[-0.0512944143707967,-0.54293181630632,0.822035880563232,0.163862555098194],[0,0,0,1],[9E+09,9E+09,9E+09,9E+09,9E+09,9E+09]];
	CONST robtarget Target_4480:=[[289.5,-239.8,-97.8],[-0.0503785277368699,-0.547513991237142,0.818991071679431,0.164146452450295],[0,0,0,1],[9E+09,9E+09,9E+09,9E+09,9E+09,9E+09]];
	CONST robtarget Target_4490:=[[284.8,-240.1,-96.6],[-0.0494516568369335,-0.552125800136082,0.815889114350191,0.164428061914728],[0,0,0,1],[9E+09,9E+09,9E+09,9E+09,9E+09,9E+09]];
	CONST robtarget Target_4500:=[[280.1,-240.4,-95.3],[-0.0485138773113708,-0.556766097158342,0.812729634716316,0.164707187509133],[0,0,0,1],[9E+09,9E+09,9E+09,9E+09,9E+09,9E+09]];
	CONST robtarget Target_4510:=[[275.4,-240.7,-94.1],[-0.0475652784406573,-0.561433672938044,0.809512308110473,0.164983630084364],[0,0,0,1],[9E+09,9E+09,9E+09,9E+09,9E+09,9E+09]];
	CONST robtarget Target_4520:=[[270.7,-241,-92.8],[-0.04657611167879,-0.566118569710976,0.806236496288795,0.165297135187669],[0,0,0,1],[9E+09,9E+09,9E+09,9E+09,9E+09,9E+09]];
	CONST robtarget Target_4530:=[[265.9,-241.2,-91.6],[-0.0455781193684878,-0.570971841278474,0.802806750959846,0.165575095093428],[0,0,0,1],[9E+09,9E+09,9E+09,9E+09,9E+09,9E+09]];
	CONST robtarget Target_4540:=[[261.2,-241.6,-90.3],[-0.044603962147879,-0.575681451164459,0.799436294963406,0.165840174991093],[0,0,0,1],[9E+09,9E+09,9E+09,9E+09,9E+09,9E+09]];
	CONST robtarget Target_4550:=[[256.5,-241.9,-89.1],[-0.0436128251589251,-0.580445150786425,0.795984264824474,0.166103577812228],[0,0,0,1],[9E+09,9E+09,9E+09,9E+09,9E+09,9E+09]];
	CONST robtarget Target_4560:=[[251.8,-242.1,-87.8],[-0.0426055282136537,-0.585257721214646,0.792452473450789,0.166364798097438],[0,0,0,1],[9E+09,9E+09,9E+09,9E+09,9E+09,9E+09]];
	CONST robtarget Target_4570:=[[247.1,-242.4,-86.6],[-0.0415634621821783,-0.590050377687373,0.788883798273689,0.166659482849602],[0,0,0,1],[9E+09,9E+09,9E+09,9E+09,9E+09,9E+09]];
	CONST robtarget Target_4580:=[[242.4,-242.7,-85.3],[-0.0405424217596268,-0.594868736122905,0.78525682561266,0.166910804473919],[0,0,0,1],[9E+09,9E+09,9E+09,9E+09,9E+09,9E+09]];
	CONST robtarget Target_4590:=[[237.6,-243,-84.1],[-0.0394894517675504,-0.599806981726168,0.781491317968587,0.167163057555683],[0,0,0,1],[9E+09,9E+09,9E+09,9E+09,9E+09,9E+09]];
	CONST robtarget Target_4600:=[[232.9,-243.3,-82.8],[-0.0384493332726948,-0.604654398226158,0.777746844476721,0.167405356494801],[0,0,0,1],[9E+09,9E+09,9E+09,9E+09,9E+09,9E+09]];
	CONST robtarget Target_4610:=[[228.2,-243.6,-81.6],[-0.0374001271246908,-0.609513532222938,0.773944668193309,0.167642879667832],[0,0,0,1],[9E+09,9E+09,9E+09,9E+09,9E+09,9E+09]];
	CONST robtarget Target_4620:=[[223.5,-243.9,-80.3],[-0.0363420920703788,-0.614382529573869,0.770085191873047,0.167875420941287],[0,0,0,1],[9E+09,9E+09,9E+09,9E+09,9E+09,9E+09]];
	CONST robtarget Target_4630:=[[218.8,-244.2,-79.1],[-0.0352789013652378,-0.61925527973127,0.766168461703898,0.168119558450798],[0,0,0,1],[9E+09,9E+09,9E+09,9E+09,9E+09,9E+09]];
	CONST robtarget Target_4640:=[[115,-250.6,-51.6],[-0.0101362950557384,-0.724712432235474,0.667264072240018,0.171603624622428],[0,0,0,1],[9E+09,9E+09,9E+09,9E+09,9E+09,9E+09]];
	CONST robtarget Target_4650:=[[110.3,-251,-50.3],[-0.00897562763950428,-0.729208103588957,0.662348090658669,0.17166824566439],[0,0,0,1],[9E+09,9E+09,9E+09,9E+09,9E+09,9E+09]];
	CONST robtarget Target_4660:=[[105.6,-251.2,-49.1],[-0.00782265456170565,-0.733639401003984,0.6574364462315,0.171724647434841],[0,0,0,1],[9E+09,9E+09,9E+09,9E+09,9E+09,9E+09]];
	CONST robtarget Target_4670:=[[100.9,-251.5,-47.8],[-0.00666858886590735,-0.738040426737729,0.652491976992652,0.171773334320405],[0,0,0,1],[9E+09,9E+09,9E+09,9E+09,9E+09,9E+09]];
	CONST robtarget Target_4680:=[[96.1,-251.8,-46.6],[-0.00549276498109347,-0.742488988783896,0.647425326252885,0.171814952765686],[0,0,0,1],[9E+09,9E+09,9E+09,9E+09,9E+09,9E+09]];
	CONST robtarget Target_4690:=[[91.4,-252.1,-45.3],[-0.00430540759594907,-0.74679156851643,0.642449494845078,0.171879211167342],[0,0,0,1],[9E+09,9E+09,9E+09,9E+09,9E+09,9E+09]];
	CONST robtarget Target_4700:=[[86.7,-252.4,-44.1],[-0.00316015182200857,-0.751051866701647,0.637459175095774,0.171921223386319],[0,0,0,1],[9E+09,9E+09,9E+09,9E+09,9E+09,9E+09]];
	CONST robtarget Target_4710:=[[82,-252.7,-42.8],[-0.00201839954074666,-0.755268500999825,0.63245758576152,0.171938418259215],[0,0,0,1],[9E+09,9E+09,9E+09,9E+09,9E+09,9E+09]];
	CONST robtarget Target_4720:=[[77.3,-253,-41.6],[-0.0008808921358361,-0.759436013773593,0.627447246685718,0.171948008535231],[0,0,0,1],[9E+09,9E+09,9E+09,9E+09,9E+09,9E+09]];
	CONST robtarget Target_4730:=[[72.6,-253.3,-40.3],[0.00025194861916876,-0.763553257561029,0.622430340887841,0.171950080349153],[0,0,0,1],[9E+09,9E+09,9E+09,9E+09,9E+09,9E+09]];
	CONST robtarget Target_4740:=[[67.8,-253.6,-39.1],[0.0014032710037228,-0.767703754987846,0.617303856271264,0.171944538850982],[0,0,0,1],[9E+09,9E+09,9E+09,9E+09,9E+09,9E+09]];
	CONST robtarget Target_4750:=[[63.1,-253.9,-37.8],[0.00252541762663588,-0.771716168657379,0.612280378113319,0.171931718644344],[0,0,0,1],[9E+09,9E+09,9E+09,9E+09,9E+09,9E+09]];
	CONST robtarget Target_4760:=[[58.4,-254.2,-36.6],[0.00368184764794892,-0.775666917664595,0.607258990533648,0.171941255243348],[0,0,0,1],[9E+09,9E+09,9E+09,9E+09,9E+09,9E+09]];
	CONST robtarget Target_4770:=[[53.7,-254.5,-35.3],[0.00479206590257211,-0.779572065269462,0.60223753104132,0.171913895195084],[0,0,0,1],[9E+09,9E+09,9E+09,9E+09,9E+09,9E+09]];
	CONST robtarget Target_4780:=[[49,-254.8,-34.1],[0.00589567441362501,-0.783422434180185,0.597220175786478,0.171879586571441],[0,0,0,1],[9E+09,9E+09,9E+09,9E+09,9E+09,9E+09]];
	CONST robtarget Target_4790:=[[44.2,-255.1,-32.8],[0.0070151140987902,-0.787295902256136,0.592104560896076,0.171837537898278],[0,0,0,1],[9E+09,9E+09,9E+09,9E+09,9E+09,9E+09]];
	CONST robtarget Target_4800:=[[39.5,-255.3,-31.6],[0.00809672271399045,-0.791007704806005,0.58713666184354,0.171789971587557],[0,0,0,1],[9E+09,9E+09,9E+09,9E+09,9E+09,9E+09]];
	CONST robtarget Target_4810:=[[34.8,-255.7,-30.3],[0.00918587623296491,-0.794714822430291,0.582109096091815,0.17173517675361],[0,0,0,1],[9E+09,9E+09,9E+09,9E+09,9E+09,9E+09]];
	CONST robtarget Target_4820:=[[30.1,-255.9,-29.1],[0.0102514536764731,-0.798311972467211,0.577166044876818,0.171674864072409],[0,0,0,1],[9E+09,9E+09,9E+09,9E+09,9E+09,9E+09]];
    !***********************************************************
    !
    ! Module:  test
    !
    ! Description:
    !   <Insert description>
    !
    ! Author: ModuleWriter
    ! Version: 1.0
    !
    !***********************************************************


